RoboDK station: ConvertMoveC.rdk

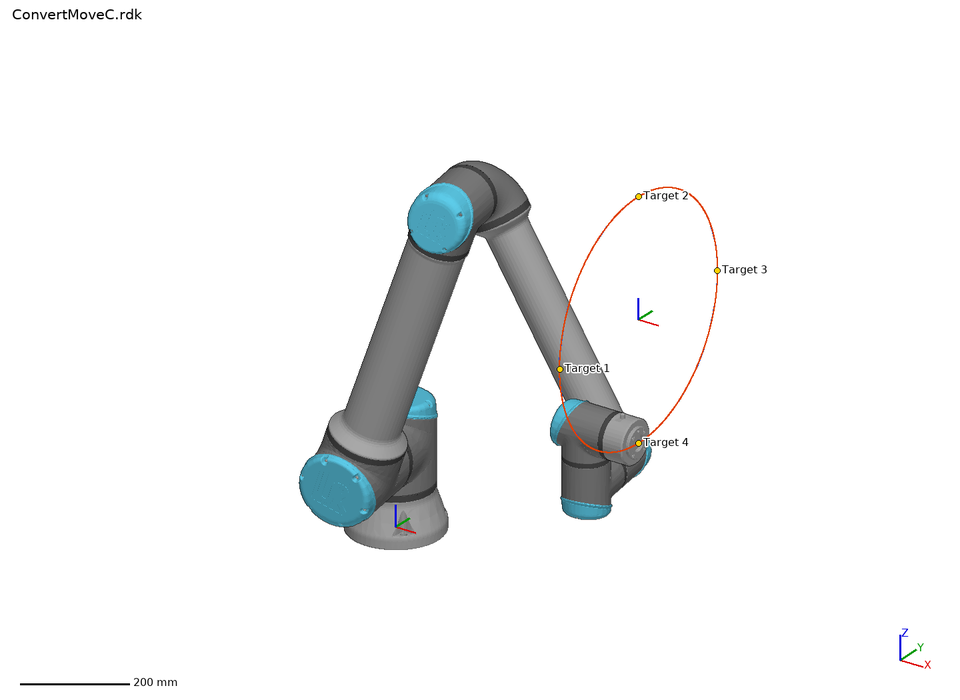
[picture v0: the station drawn from its stored meshes, robots at their saved joint values, targets as dots, program paths as lines]
Station ConvertMoveC (saved by RoboDK 5.5.2). Poses are relative to the parent item; angles as X-Y-Z fixed-axis rotations.
Station parameters (name, value as stored): ProgUtilities-Settings
  - frame UR10e Base at (0, 0, 0) mm
    - robot UR10e: 6 axes, payload 10 kg, reach 1300 mm, repeatability 0.05 mm, weight 28.9 kg
        modified DH rows (alpha deg, a mm, theta deg, d mm): 0, 0, 0, 180.7; 90, 0, 180, 0; 0, 612.6, 0, 0; 0, 571.335, 0, 174.15; -90, 0, 0, 119.85; 90, 0, 180, 116.55
        joint limits [-360, -360, -360, -360, -360, -360] to [360, 360, 360, 360, 360, 360]; home [0, -90, -90, 0, 90, 0]; saved at [8.78, -108.762, -132.424, 61.186, 81.22, 0]
    - frame Frame 2 at (610, -100, 630) mm
      - target Target 1 (Cartesian target) at (0, -250, 0) mm, rotated rx -90 ry 0 rz -90 deg; joints [-18.618, -97.519, -111.584, 29.103, 108.618, 0] of UR10e
      - target Target 2 (Cartesian target) at (0, 0, 250) mm, rotated rx -90 ry 0 rz -90 deg; joints [8.78, -80.759, -101.769, 2.528, 81.22, 0] of UR10e
      - target Target 3 (Cartesian target) at (0, 250, 0) mm, rotated rx -90 ry 0 rz -90 deg; joints [36.643, -88.986, -120.711, 29.698, 53.357, 0] of UR10e
      - target Target 4 (Cartesian target) at (0, 0, -250) mm, rotated rx -90 ry 0 rz -90 deg; joints [8.78, -108.762, -132.424, 61.186, 81.22, 0] of UR10e
  - program Prog1 (4 instructions, listed below)
  - program Prog1 Linear MoveC (1580 instructions, listed below)
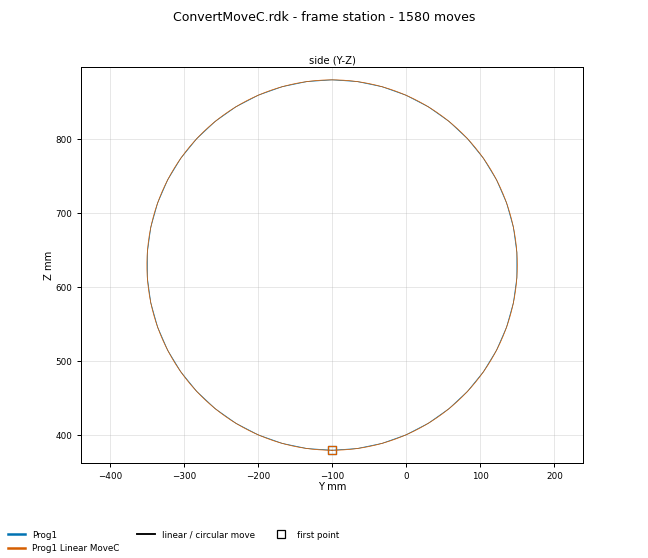
[picture p0: tool path of ConvertMoveC.rdk in frame station, 1580 of 1580 moves have a stored position in this frame; points joined in program order, loops and branches not executed]

--- program Prog1 (robot UR10e) ---
  Set Ref.: Frame 2
  MoveJ (Target 4)
  MoveC (Target 1, Target 2)
  MoveC (Target 3, Target 4)

--- program Prog1 Linear MoveC (robot UR10e) ---
  Set Ref.: Frame 2
  MoveJ (Target 4) to (0, 0, -250) mm, rotated rx -90 ry 0 rz -90 deg; joints [8.78, -108.762, -132.424, 61.186, 81.22, 0]
  MoveC (Target 1, Target 2)
  MoveL 3 to (0, 0, -250) mm, rotated rx -90 ry 0 rz -90 deg; joints [8.78, -108.762, -132.424, 61.186, 81.22, 0]
  MoveL 4 to (0, 0, -250) mm, rotated rx -90 ry 0 rz -90 deg; joints [8.78, -108.762, -132.424, 61.186, 81.22, 0]
  MoveL 5 to (0, -1, -250) mm, rotated rx -90 ry 0 rz -90 deg; joints [8.66, -108.775, -132.401, 61.176, 81.34, 0]
  MoveL 6 to (0, -2, -249.99) mm, rotated rx -90 ry 0 rz -90 deg; joints [8.541, -108.787, -132.379, 61.166, 81.459, 0]
  MoveL 7 to (0, -3, -249.98) mm, rotated rx -90 ry 0 rz -90 deg; joints [8.421, -108.8, -132.356, 61.156, 81.579, 0]
  MoveL 8 to (0, -4, -249.97) mm, rotated rx -90 ry 0 rz -90 deg; joints [8.301, -108.811, -132.333, 61.144, 81.699, 0]
  MoveL 9 to (0, -5, -249.95) mm, rotated rx -90 ry 0 rz -90 deg; joints [8.182, -108.823, -132.309, 61.132, 81.819, 0]
  MoveL 10 to (0, -5.99, -249.93) mm, rotated rx -90 ry 0 rz -90 deg; joints [8.062, -108.834, -132.286, 61.12, 81.938, 0]
  MoveL 11 to (0, -6.99, -249.9) mm, rotated rx -90 ry 0 rz -90 deg; joints [7.942, -108.845, -132.262, 61.107, 82.058, 0]
  MoveL 12 to (0, -7.99, -249.87) mm, rotated rx -90 ry 0 rz -90 deg; joints [7.823, -108.855, -132.237, 61.093, 82.177, 0]
  MoveL 13 to (0, -8.99, -249.84) mm, rotated rx -90 ry 0 rz -90 deg; joints [7.703, -108.866, -132.213, 61.078, 82.297, 0]
  MoveL 14 to (0, -9.99, -249.8) mm, rotated rx -90 ry 0 rz -90 deg; joints [7.584, -108.875, -132.188, 61.063, 82.416, 0]
  MoveL 15 to (0, -10.99, -249.76) mm, rotated rx -90 ry 0 rz -90 deg; joints [7.464, -108.885, -132.163, 61.048, 82.536, 0]
  MoveL 16 to (0, -11.99, -249.71) mm, rotated rx -90 ry 0 rz -90 deg; joints [7.345, -108.894, -132.138, 61.032, 82.655, 0]
  MoveL 17 to (0, -12.98, -249.66) mm, rotated rx -90 ry 0 rz -90 deg; joints [7.225, -108.903, -132.112, 61.015, 82.775, 0]
  MoveL 18 to (0, -13.98, -249.61) mm, rotated rx -90 ry 0 rz -90 deg; joints [7.106, -108.912, -132.086, 60.998, 82.894, 0]
  MoveL 19 to (0, -14.98, -249.55) mm, rotated rx -90 ry 0 rz -90 deg; joints [6.987, -108.92, -132.06, 60.98, 83.013, 0]
  MoveL 20 to (0, -15.98, -249.49) mm, rotated rx -90 ry 0 rz -90 deg; joints [6.868, -108.928, -132.033, 60.961, 83.132, 0]
  MoveL 21 to (0, -16.97, -249.42) mm, rotated rx -90 ry 0 rz -90 deg; joints [6.749, -108.936, -132.007, 60.942, 83.251, 0]
  MoveL 22 to (0, -17.97, -249.35) mm, rotated rx -90 ry 0 rz -90 deg; joints [6.629, -108.943, -131.98, 60.923, 83.371, 0]
  MoveL 23 to (0, -18.97, -249.28) mm, rotated rx -90 ry 0 rz -90 deg; joints [6.51, -108.95, -131.952, 60.902, 83.49, 0]
  MoveL 24 to (0, -19.96, -249.2) mm, rotated rx -90 ry 0 rz -90 deg; joints [6.392, -108.957, -131.925, 60.881, 83.608, 0]
  MoveL 25 to (0, -20.96, -249.12) mm, rotated rx -90 ry 0 rz -90 deg; joints [6.273, -108.963, -131.897, 60.86, 83.727, 0]
  MoveL 26 to (0, -21.95, -249.03) mm, rotated rx -90 ry 0 rz -90 deg; joints [6.154, -108.969, -131.869, 60.838, 83.846, 0]
  MoveL 27 to (0, -22.95, -248.94) mm, rotated rx -90 ry 0 rz -90 deg; joints [6.035, -108.975, -131.84, 60.815, 83.965, 0]
  MoveL 28 to (0, -23.94, -248.85) mm, rotated rx -90 ry 0 rz -90 deg; joints [5.917, -108.981, -131.812, 60.792, 84.083, 0]
  MoveL 29 to (0, -24.94, -248.75) mm, rotated rx -90 ry 0 rz -90 deg; joints [5.798, -108.986, -131.783, 60.769, 84.202, 0]
  MoveL 30 to (0, -25.93, -248.65) mm, rotated rx -90 ry 0 rz -90 deg; joints [5.68, -108.991, -131.754, 60.744, 84.32, 0]
  MoveL 31 to (0, -26.93, -248.55) mm, rotated rx -90 ry 0 rz -90 deg; joints [5.561, -108.995, -131.724, 60.719, 84.439, 0]
  MoveL 32 to (0, -27.92, -248.44) mm, rotated rx -90 ry 0 rz -90 deg; joints [5.443, -108.999, -131.695, 60.694, 84.557, 0]
  MoveL 33 to (0, -28.91, -248.32) mm, rotated rx -90 ry 0 rz -90 deg; joints [5.325, -109.003, -131.665, 60.668, 84.675, 0]
  MoveL 34 to (0, -29.91, -248.2) mm, rotated rx -90 ry 0 rz -90 deg; joints [5.207, -109.007, -131.634, 60.641, 84.793, 0]
  MoveL 35 to (0, -30.9, -248.08) mm, rotated rx -90 ry 0 rz -90 deg; joints [5.089, -109.01, -131.604, 60.614, 84.911, 0]
  MoveL 36 to (0, -31.89, -247.96) mm, rotated rx -90 ry 0 rz -90 deg; joints [4.971, -109.013, -131.573, 60.586, 85.029, 0]
  MoveL 37 to (0, -32.88, -247.83) mm, rotated rx -90 ry 0 rz -90 deg; joints [4.853, -109.016, -131.542, 60.558, 85.147, 0]
  MoveL 38 to (0, -33.87, -247.7) mm, rotated rx -90 ry 0 rz -90 deg; joints [4.736, -109.018, -131.511, 60.529, 85.265, 0]
  MoveL 39 to (0, -34.86, -247.56) mm, rotated rx -90 ry 0 rz -90 deg; joints [4.618, -109.02, -131.479, 60.5, 85.382, 0]
  MoveL 40 to (0, -35.85, -247.42) mm, rotated rx -90 ry 0 rz -90 deg; joints [4.501, -109.022, -131.448, 60.47, 85.499, 0]
  MoveL 41 to (0, -36.84, -247.27) mm, rotated rx -90 ry 0 rz -90 deg; joints [4.383, -109.023, -131.415, 60.439, 85.617, 0]
  MoveL 42 to (0, -37.83, -247.12) mm, rotated rx -90 ry 0 rz -90 deg; joints [4.266, -109.025, -131.383, 60.408, 85.734, 0]
  MoveL 43 to (0, -38.81, -246.97) mm, rotated rx -90 ry 0 rz -90 deg; joints [4.149, -109.025, -131.351, 60.376, 85.851, 0]
  MoveL 44 to (0, -39.8, -246.81) mm, rotated rx -90 ry 0 rz -90 deg; joints [4.032, -109.026, -131.318, 60.344, 85.968, 0]
  MoveL 45 to (0, -40.79, -246.65) mm, rotated rx -90 ry 0 rz -90 deg; joints [3.915, -109.026, -131.285, 60.311, 86.085, 0]
  MoveL 46 to (0, -41.77, -246.49) mm, rotated rx -90 ry 0 rz -90 deg; joints [3.799, -109.026, -131.251, 60.278, 86.201, 0]
  MoveL 47 to (0, -42.76, -246.32) mm, rotated rx -90 ry 0 rz -90 deg; joints [3.682, -109.026, -131.218, 60.244, 86.318, 0]
  MoveL 48 to (0, -43.74, -246.14) mm, rotated rx -90 ry 0 rz -90 deg; joints [3.566, -109.025, -131.184, 60.209, 86.434, 0]
  MoveL 49 to (0, -44.72, -245.97) mm, rotated rx -90 ry 0 rz -90 deg; joints [3.449, -109.024, -131.15, 60.174, 86.551, 0]
  MoveL 50 to (0, -45.71, -245.79) mm, rotated rx -90 ry 0 rz -90 deg; joints [3.333, -109.023, -131.116, 60.139, 86.667, 0]
  MoveL 51 to (0, -46.69, -245.6) mm, rotated rx -90 ry 0 rz -90 deg; joints [3.217, -109.021, -131.081, 60.103, 86.783, 0]
  MoveL 52 to (0, -47.67, -245.41) mm, rotated rx -90 ry 0 rz -90 deg; joints [3.101, -109.02, -131.046, 60.066, 86.899, 0]
  MoveL 53 to (0, -48.65, -245.22) mm, rotated rx -90 ry 0 rz -90 deg; joints [2.986, -109.017, -131.011, 60.029, 87.014, 0]
  MoveL 54 to (0, -49.63, -245.02) mm, rotated rx -90 ry 0 rz -90 deg; joints [2.87, -109.015, -130.976, 59.991, 87.13, 0]
  MoveL 55 to (0, -50.61, -244.82) mm, rotated rx -90 ry 0 rz -90 deg; joints [2.755, -109.012, -130.941, 59.953, 87.245, 0]
  MoveL 56 to (0, -51.59, -244.62) mm, rotated rx -90 ry 0 rz -90 deg; joints [2.639, -109.009, -130.905, 59.914, 87.361, 0]
  MoveL 57 to (0, -52.56, -244.41) mm, rotated rx -90 ry 0 rz -90 deg; joints [2.524, -109.006, -130.869, 59.875, 87.476, 0]
  MoveL 58 to (0, -53.54, -244.2) mm, rotated rx -90 ry 0 rz -90 deg; joints [2.409, -109.002, -130.833, 59.835, 87.591, 0]
  MoveL 59 to (0, -54.52, -243.98) mm, rotated rx -90 ry 0 rz -90 deg; joints [2.295, -108.999, -130.796, 59.795, 87.705, 0]
  MoveL 60 to (0, -55.49, -243.76) mm, rotated rx -90 ry 0 rz -90 deg; joints [2.18, -108.994, -130.759, 59.754, 87.82, 0]
  MoveL 61 to (0, -56.46, -243.54) mm, rotated rx -90 ry 0 rz -90 deg; joints [2.066, -108.99, -130.722, 59.712, 87.934, 0]
  MoveL 62 to (0, -57.44, -243.31) mm, rotated rx -90 ry 0 rz -90 deg; joints [1.951, -108.985, -130.685, 59.67, 88.049, 0]
  MoveL 63 to (0, -58.41, -243.08) mm, rotated rx -90 ry 0 rz -90 deg; joints [1.837, -108.98, -130.648, 59.628, 88.163, 0]
  MoveL 64 to (0, -59.38, -242.85) mm, rotated rx -90 ry 0 rz -90 deg; joints [1.723, -108.975, -130.61, 59.585, 88.277, 0]
  MoveL 65 to (0, -60.35, -242.61) mm, rotated rx -90 ry 0 rz -90 deg; joints [1.61, -108.969, -130.572, 59.541, 88.39, 0]
  MoveL 66 to (0, -61.32, -242.36) mm, rotated rx -90 ry 0 rz -90 deg; joints [1.496, -108.963, -130.534, 59.497, 88.504, 0]
  MoveL 67 to (0, -62.29, -242.12) mm, rotated rx -90 ry 0 rz -90 deg; joints [1.383, -108.957, -130.496, 59.453, 88.617, 0]
  MoveL 68 to (0, -63.26, -241.87) mm, rotated rx -90 ry 0 rz -90 deg; joints [1.27, -108.951, -130.457, 59.408, 88.73, 0]
  MoveL 69 to (0, -64.22, -241.61) mm, rotated rx -90 ry 0 rz -90 deg; joints [1.157, -108.944, -130.418, 59.362, 88.843, 0]
  MoveL 70 to (0, -65.19, -241.35) mm, rotated rx -90 ry 0 rz -90 deg; joints [1.044, -108.937, -130.379, 59.316, 88.956, 0]
  MoveL 71 to (0, -66.15, -241.09) mm, rotated rx -90 ry 0 rz -90 deg; joints [0.931, -108.93, -130.34, 59.27, 89.069, 0]
  MoveL 72 to (0, -67.11, -240.82) mm, rotated rx -90 ry 0 rz -90 deg; joints [0.819, -108.922, -130.3, 59.222, 89.181, 0]
  MoveL 73 to (0, -68.08, -240.55) mm, rotated rx -90 ry 0 rz -90 deg; joints [0.707, -108.914, -130.261, 59.175, 89.293, 0]
  MoveL 74 to (0, -69.04, -240.28) mm, rotated rx -90 ry 0 rz -90 deg; joints [0.595, -108.906, -130.221, 59.127, 89.405, 0]
  MoveL 75 to (0, -70, -240) mm, rotated rx -90 ry 0 rz -90 deg; joints [0.483, -108.898, -130.18, 59.078, 89.517, 0]
  MoveL 76 to (0, -70.96, -239.72) mm, rotated rx -90 ry 0 rz -90 deg; joints [0.371, -108.889, -130.14, 59.029, 89.629, 0]
  MoveL 77 to (0, -71.91, -239.43) mm, rotated rx -90 ry 0 rz -90 deg; joints [0.26, -108.88, -130.099, 58.98, 89.74, 0]
  MoveL 78 to (0, -72.87, -239.14) mm, rotated rx -90 ry 0 rz -90 deg; joints [0.149, -108.871, -130.059, 58.929, 89.851, 0]
  MoveL 79 to (0, -73.83, -238.85) mm, rotated rx -90 ry 0 rz -90 deg; joints [0.038, -108.861, -130.017, 58.879, 89.962, 0]
  MoveL 80 to (0, -74.78, -238.55) mm, rotated rx -90 ry 0 rz -90 deg; joints [-0.073, -108.852, -129.976, 58.828, 90.073, 0]
  MoveL 81 to (0, -75.73, -238.25) mm, rotated rx -90 ry 0 rz -90 deg; joints [-0.184, -108.842, -129.935, 58.776, 90.184, 0]
  MoveL 82 to (0, -76.68, -237.95) mm, rotated rx -90 ry 0 rz -90 deg; joints [-0.294, -108.831, -129.893, 58.724, 90.294, 0]
  MoveL 83 to (0, -77.63, -237.64) mm, rotated rx -90 ry 0 rz -90 deg; joints [-0.404, -108.821, -129.851, 58.672, 90.404, 0]
  MoveL 84 to (0, -78.58, -237.33) mm, rotated rx -90 ry 0 rz -90 deg; joints [-0.514, -108.81, -129.809, 58.619, 90.514, 0]
  MoveL 85 to (0, -79.53, -237.01) mm, rotated rx -90 ry 0 rz -90 deg; joints [-0.624, -108.799, -129.766, 58.565, 90.624, 0]
  MoveL 86 to (0, -80.48, -236.69) mm, rotated rx -90 ry 0 rz -90 deg; joints [-0.733, -108.788, -129.724, 58.511, 90.733, 0]
  MoveL 87 to (0, -81.42, -236.37) mm, rotated rx -90 ry 0 rz -90 deg; joints [-0.842, -108.776, -129.681, 58.457, 90.842, 0]
  MoveL 88 to (0, -82.37, -236.04) mm, rotated rx -90 ry 0 rz -90 deg; joints [-0.951, -108.764, -129.638, 58.402, 90.951, 0]
  MoveL 89 to (0, -83.31, -235.71) mm, rotated rx -90 ry 0 rz -90 deg; joints [-1.06, -108.752, -129.595, 58.347, 91.06, 0]
  MoveL 90 to (0, -84.25, -235.38) mm, rotated rx -90 ry 0 rz -90 deg; joints [-1.169, -108.74, -129.551, 58.291, 91.169, 0]
  MoveL 91 to (0, -85.19, -235.04) mm, rotated rx -90 ry 0 rz -90 deg; joints [-1.277, -108.727, -129.508, 58.235, 91.277, 0]
  MoveL 92 to (0, -86.13, -234.69) mm, rotated rx -90 ry 0 rz -90 deg; joints [-1.385, -108.714, -129.464, 58.178, 91.385, 0]
  MoveL 93 to (0, -87.07, -234.35) mm, rotated rx -90 ry 0 rz -90 deg; joints [-1.493, -108.701, -129.42, 58.121, 91.493, 0]
  MoveL 94 to (0, -88, -234) mm, rotated rx -90 ry 0 rz -90 deg; joints [-1.6, -108.687, -129.376, 58.063, 91.6, 0]
  MoveL 95 to (0, -88.94, -233.64) mm, rotated rx -90 ry 0 rz -90 deg; joints [-1.708, -108.674, -129.331, 58.005, 91.708, 0]
  MoveL 96 to (0, -89.87, -233.29) mm, rotated rx -90 ry 0 rz -90 deg; joints [-1.815, -108.66, -129.287, 57.946, 91.815, 0]
  MoveL 97 to (0, -90.8, -232.93) mm, rotated rx -90 ry 0 rz -90 deg; joints [-1.922, -108.646, -129.242, 57.887, 91.922, 0]
  MoveL 98 to (0, -91.73, -232.56) mm, rotated rx -90 ry 0 rz -90 deg; joints [-2.028, -108.631, -129.197, 57.828, 92.028, 0]
  MoveL 99 to (0, -92.66, -232.19) mm, rotated rx -90 ry 0 rz -90 deg; joints [-2.135, -108.617, -129.151, 57.768, 92.135, 0]
  MoveL 100 to (0, -93.59, -231.82) mm, rotated rx -90 ry 0 rz -90 deg; joints [-2.241, -108.602, -129.106, 57.708, 92.241, 0]
  MoveL 101 to (0, -94.52, -231.44) mm, rotated rx -90 ry 0 rz -90 deg; joints [-2.346, -108.587, -129.06, 57.647, 92.346, 0]
  MoveL 102 to (0, -95.44, -231.07) mm, rotated rx -90 ry 0 rz -90 deg; joints [-2.452, -108.571, -129.014, 57.586, 92.452, 0]
  MoveL 103 to (0, -96.36, -230.68) mm, rotated rx -90 ry 0 rz -90 deg; joints [-2.557, -108.555, -128.968, 57.524, 92.557, 0]
  MoveL 104 to (0, -97.28, -230.3) mm, rotated rx -90 ry 0 rz -90 deg; joints [-2.662, -108.54, -128.922, 57.462, 92.662, 0]
  MoveL 105 to (0, -98.2, -229.9) mm, rotated rx -90 ry 0 rz -90 deg; joints [-2.767, -108.523, -128.876, 57.399, 92.767, 0]
  MoveL 106 to (0, -99.12, -229.51) mm, rotated rx -90 ry 0 rz -90 deg; joints [-2.872, -108.507, -128.829, 57.336, 92.872, 0]
  MoveL 107 to (0, -100.04, -229.11) mm, rotated rx -90 ry 0 rz -90 deg; joints [-2.976, -108.49, -128.782, 57.273, 92.976, 0]
  MoveL 108 to (0, -100.95, -228.71) mm, rotated rx -90 ry 0 rz -90 deg; joints [-3.08, -108.474, -128.735, 57.209, 93.08, 0]
  MoveL 109 to (0, -101.87, -228.31) mm, rotated rx -90 ry 0 rz -90 deg; joints [-3.184, -108.456, -128.688, 57.145, 93.184, 0]
  MoveL 110 to (0, -102.78, -227.9) mm, rotated rx -90 ry 0 rz -90 deg; joints [-3.287, -108.439, -128.641, 57.08, 93.287, 0]
  MoveL 111 to (0, -103.69, -227.48) mm, rotated rx -90 ry 0 rz -90 deg; joints [-3.39, -108.422, -128.593, 57.015, 93.39, 0]
  MoveL 112 to (0, -104.6, -227.07) mm, rotated rx -90 ry 0 rz -90 deg; joints [-3.493, -108.404, -128.546, 56.949, 93.493, 0]
  MoveL 113 to (0, -105.5, -226.65) mm, rotated rx -90 ry 0 rz -90 deg; joints [-3.596, -108.386, -128.498, 56.883, 93.596, 0]
  MoveL 114 to (0, -106.41, -226.22) mm, rotated rx -90 ry 0 rz -90 deg; joints [-3.698, -108.367, -128.45, 56.817, 93.698, 0]
  MoveL 115 to (0, -107.31, -225.8) mm, rotated rx -90 ry 0 rz -90 deg; joints [-3.8, -108.349, -128.401, 56.75, 93.8, 0]
  MoveL 116 to (0, -108.21, -225.37) mm, rotated rx -90 ry 0 rz -90 deg; joints [-3.902, -108.33, -128.353, 56.683, 93.902, 0]
  MoveL 117 to (0, -109.11, -224.93) mm, rotated rx -90 ry 0 rz -90 deg; joints [-4.004, -108.311, -128.304, 56.615, 94.004, 0]
  MoveL 118 to (0, -110.01, -224.49) mm, rotated rx -90 ry 0 rz -90 deg; joints [-4.105, -108.292, -128.255, 56.547, 94.105, 0]
  MoveL 119 to (0, -110.91, -224.05) mm, rotated rx -90 ry 0 rz -90 deg; joints [-4.206, -108.273, -128.206, 56.479, 94.206, 0]
  MoveL 120 to (0, -111.8, -223.61) mm, rotated rx -90 ry 0 rz -90 deg; joints [-4.307, -108.253, -128.157, 56.41, 94.307, 0]
  MoveL 121 to (0, -112.7, -223.16) mm, rotated rx -90 ry 0 rz -90 deg; joints [-4.407, -108.233, -128.108, 56.341, 94.407, 0]
  MoveL 122 to (0, -113.59, -222.71) mm, rotated rx -90 ry 0 rz -90 deg; joints [-4.507, -108.213, -128.058, 56.271, 94.507, 0]
  MoveL 123 to (0, -114.48, -222.25) mm, rotated rx -90 ry 0 rz -90 deg; joints [-4.607, -108.193, -128.009, 56.201, 94.607, 0]
  MoveL 124 to (0, -115.36, -221.79) mm, rotated rx -90 ry 0 rz -90 deg; joints [-4.706, -108.172, -127.959, 56.131, 94.706, 0]
  MoveL 125 to (0, -116.25, -221.33) mm, rotated rx -90 ry 0 rz -90 deg; joints [-4.806, -108.151, -127.909, 56.06, 94.806, 0]
  MoveL 126 to (0, -117.13, -220.86) mm, rotated rx -90 ry 0 rz -90 deg; joints [-4.905, -108.13, -127.859, 55.989, 94.905, 0]
  MoveL 127 to (0, -118.01, -220.39) mm, rotated rx -90 ry 0 rz -90 deg; joints [-5.003, -108.109, -127.808, 55.917, 95.003, 0]
  MoveL 128 to (0, -118.89, -219.92) mm, rotated rx -90 ry 0 rz -90 deg; joints [-5.101, -108.088, -127.758, 55.846, 95.101, 0]
  MoveL 129 to (0, -119.77, -219.44) mm, rotated rx -90 ry 0 rz -90 deg; joints [-5.199, -108.066, -127.707, 55.773, 95.2, 0]
  MoveL 130 to (0, -120.65, -218.96) mm, rotated rx -90 ry 0 rz -90 deg; joints [-5.297, -108.044, -127.656, 55.701, 95.297, 0]
  MoveL 131 to (0, -121.52, -218.48) mm, rotated rx -90 ry 0 rz -90 deg; joints [-5.395, -108.022, -127.605, 55.627, 95.395, 0]
  MoveL 132 to (0, -122.39, -217.99) mm, rotated rx -90 ry 0 rz -90 deg; joints [-5.492, -108, -127.554, 55.554, 95.492, 0]
  MoveL 133 to (0, -123.27, -217.5) mm, rotated rx -90 ry 0 rz -90 deg; joints [-5.589, -107.978, -127.503, 55.48, 95.589, 0]
  MoveL 134 to (0, -124.13, -217) mm, rotated rx -90 ry 0 rz -90 deg; joints [-5.685, -107.955, -127.451, 55.406, 95.685, 0]
  MoveL 135 to (0, -125, -216.51) mm, rotated rx -90 ry 0 rz -90 deg; joints [-5.781, -107.932, -127.399, 55.331, 95.781, 0]
  MoveL 136 to (0, -125.86, -216.01) mm, rotated rx -90 ry 0 rz -90 deg; joints [-5.877, -107.909, -127.348, 55.256, 95.877, 0]
  MoveL 137 to (0, -126.73, -215.5) mm, rotated rx -90 ry 0 rz -90 deg; joints [-5.973, -107.886, -127.296, 55.181, 95.973, 0]
  MoveL 138 to (0, -127.59, -214.99) mm, rotated rx -90 ry 0 rz -90 deg; joints [-6.068, -107.862, -127.243, 55.106, 96.068, 0]
  MoveL 139 to (0, -128.45, -214.48) mm, rotated rx -90 ry 0 rz -90 deg; joints [-6.163, -107.838, -127.191, 55.03, 96.163, 0]
  MoveL 140 to (0, -129.3, -213.97) mm, rotated rx -90 ry 0 rz -90 deg; joints [-6.258, -107.815, -127.139, 54.953, 96.258, 0]
  MoveL 141 to (0, -130.16, -213.45) mm, rotated rx -90 ry 0 rz -90 deg; joints [-6.352, -107.79, -127.086, 54.876, 96.352, 0]
  MoveL 142 to (0, -131.01, -212.92) mm, rotated rx -90 ry 0 rz -90 deg; joints [-6.446, -107.766, -127.033, 54.799, 96.446, 0]
  MoveL 143 to (0, -131.86, -212.4) mm, rotated rx -90 ry 0 rz -90 deg; joints [-6.54, -107.742, -126.98, 54.722, 96.54, 0]
  MoveL 144 to (0, -132.71, -211.87) mm, rotated rx -90 ry 0 rz -90 deg; joints [-6.633, -107.717, -126.927, 54.644, 96.633, 0]
  MoveL 145 to (0, -133.55, -211.34) mm, rotated rx -90 ry 0 rz -90 deg; joints [-6.726, -107.692, -126.874, 54.566, 96.726, 0]
  MoveL 146 to (0, -134.4, -210.8) mm, rotated rx -90 ry 0 rz -90 deg; joints [-6.819, -107.667, -126.821, 54.488, 96.819, 0]
  MoveL 147 to (0, -135.24, -210.26) mm, rotated rx -90 ry 0 rz -90 deg; joints [-6.911, -107.642, -126.767, 54.409, 96.911, 0]
  MoveL 148 to (0, -136.08, -209.72) mm, rotated rx -90 ry 0 rz -90 deg; joints [-7.003, -107.616, -126.714, 54.33, 97.003, 0]
  MoveL 149 to (0, -136.91, -209.18) mm, rotated rx -90 ry 0 rz -90 deg; joints [-7.095, -107.59, -126.66, 54.25, 97.095, 0]
  MoveL 150 to (0, -137.75, -208.63) mm, rotated rx -90 ry 0 rz -90 deg; joints [-7.187, -107.565, -126.606, 54.171, 97.187, 0]
  MoveL 151 to (0, -138.58, -208.08) mm, rotated rx -90 ry 0 rz -90 deg; joints [-7.278, -107.538, -126.552, 54.09, 97.278, 0]
  MoveL 152 to (0, -139.41, -207.52) mm, rotated rx -90 ry 0 rz -90 deg; joints [-7.368, -107.512, -126.498, 54.01, 97.368, 0]
  MoveL 153 to (0, -140.24, -206.96) mm, rotated rx -90 ry 0 rz -90 deg; joints [-7.459, -107.486, -126.443, 53.929, 97.459, 0]
  MoveL 154 to (0, -141.07, -206.4) mm, rotated rx -90 ry 0 rz -90 deg; joints [-7.549, -107.459, -126.389, 53.848, 97.549, 0]
  MoveL 155 to (0, -141.89, -205.83) mm, rotated rx -90 ry 0 rz -90 deg; joints [-7.639, -107.432, -126.334, 53.767, 97.639, 0]
  MoveL 156 to (0, -142.71, -205.26) mm, rotated rx -90 ry 0 rz -90 deg; joints [-7.728, -107.405, -126.279, 53.685, 97.728, 0]
  MoveL 157 to (0, -143.53, -204.69) mm, rotated rx -90 ry 0 rz -90 deg; joints [-7.817, -107.378, -126.225, 53.603, 97.817, 0]
  MoveL 158 to (0, -144.35, -204.12) mm, rotated rx -90 ry 0 rz -90 deg; joints [-7.906, -107.351, -126.17, 53.52, 97.906, 0]
  MoveL 159 to (0, -145.16, -203.54) mm, rotated rx -90 ry 0 rz -90 deg; joints [-7.995, -107.323, -126.114, 53.438, 97.995, 0]
  MoveL 160 to (0, -145.97, -202.96) mm, rotated rx -90 ry 0 rz -90 deg; joints [-8.083, -107.295, -126.059, 53.355, 98.083, 0]
  MoveL 161 to (0, -146.78, -202.37) mm, rotated rx -90 ry 0 rz -90 deg; joints [-8.171, -107.268, -126.004, 53.271, 98.171, 0]
  MoveL 162 to (0, -147.59, -201.78) mm, rotated rx -90 ry 0 rz -90 deg; joints [-8.258, -107.239, -125.948, 53.188, 98.258, 0]
  MoveL 163 to (0, -148.4, -201.19) mm, rotated rx -90 ry 0 rz -90 deg; joints [-8.345, -107.211, -125.892, 53.104, 98.345, 0]
  MoveL 164 to (0, -149.2, -200.6) mm, rotated rx -90 ry 0 rz -90 deg; joints [-8.432, -107.183, -125.837, 53.019, 98.432, 0]
  MoveL 165 to (0, -150, -200) mm, rotated rx -90 ry 0 rz -90 deg; joints [-8.518, -107.154, -125.781, 52.935, 98.518, 0]
  MoveL 166 to (0, -150.8, -199.4) mm, rotated rx -90 ry 0 rz -90 deg; joints [-8.605, -107.125, -125.725, 52.85, 98.605, 0]
  MoveL 167 to (0, -151.6, -198.79) mm, rotated rx -90 ry 0 rz -90 deg; joints [-8.69, -107.096, -125.669, 52.765, 98.69, 0]
  MoveL 168 to (0, -152.39, -198.19) mm, rotated rx -90 ry 0 rz -90 deg; joints [-8.776, -107.067, -125.612, 52.68, 98.776, 0]
  MoveL 169 to (0, -153.18, -197.58) mm, rotated rx -90 ry 0 rz -90 deg; joints [-8.861, -107.038, -125.556, 52.594, 98.861, 0]
  MoveL 170 to (0, -153.97, -196.96) mm, rotated rx -90 ry 0 rz -90 deg; joints [-8.945, -107.008, -125.499, 52.508, 98.946, 0]
  MoveL 171 to (0, -154.75, -196.34) mm, rotated rx -90 ry 0 rz -90 deg; joints [-9.03, -106.979, -125.443, 52.421, 99.03, 0]
  MoveL 172 to (0, -155.54, -195.72) mm, rotated rx -90 ry 0 rz -90 deg; joints [-9.114, -106.949, -125.386, 52.335, 99.114, 0]
  MoveL 173 to (0, -156.32, -195.1) mm, rotated rx -90 ry 0 rz -90 deg; joints [-9.198, -106.919, -125.329, 52.248, 99.198, 0]
  MoveL 174 to (0, -157.1, -194.48) mm, rotated rx -90 ry 0 rz -90 deg; joints [-9.281, -106.889, -125.272, 52.161, 99.281, 0]
  MoveL 175 to (0, -157.87, -193.85) mm, rotated rx -90 ry 0 rz -90 deg; joints [-9.364, -106.859, -125.215, 52.073, 99.364, 0]
  MoveL 176 to (0, -158.65, -193.21) mm, rotated rx -90 ry 0 rz -90 deg; joints [-9.447, -106.828, -125.158, 51.986, 99.447, 0]
  MoveL 177 to (0, -159.42, -192.58) mm, rotated rx -90 ry 0 rz -90 deg; joints [-9.529, -106.797, -125.1, 51.898, 99.529, 0]
  MoveL 178 to (0, -160.19, -191.94) mm, rotated rx -90 ry 0 rz -90 deg; joints [-9.611, -106.767, -125.043, 51.809, 99.611, 0]
  MoveL 179 to (0, -160.95, -191.3) mm, rotated rx -90 ry 0 rz -90 deg; joints [-9.692, -106.736, -124.985, 51.721, 99.692, 0]
  MoveL 180 to (0, -161.72, -190.65) mm, rotated rx -90 ry 0 rz -90 deg; joints [-9.774, -106.705, -124.928, 51.632, 99.774, 0]
  MoveL 181 to (0, -162.48, -190) mm, rotated rx -90 ry 0 rz -90 deg; joints [-9.855, -106.673, -124.87, 51.543, 99.855, 0]
  MoveL 182 to (0, -163.23, -189.35) mm, rotated rx -90 ry 0 rz -90 deg; joints [-9.935, -106.642, -124.812, 51.454, 99.935, 0]
  MoveL 183 to (0, -163.99, -188.7) mm, rotated rx -90 ry 0 rz -90 deg; joints [-10.015, -106.61, -124.754, 51.364, 100.015, 0]
  MoveL 184 to (0, -164.74, -188.04) mm, rotated rx -90 ry 0 rz -90 deg; joints [-10.095, -106.578, -124.696, 51.274, 100.095, 0]
  MoveL 185 to (0, -165.49, -187.38) mm, rotated rx -90 ry 0 rz -90 deg; joints [-10.175, -106.547, -124.638, 51.184, 100.175, 0]
  MoveL 186 to (0, -166.24, -186.72) mm, rotated rx -90 ry 0 rz -90 deg; joints [-10.254, -106.514, -124.579, 51.094, 100.254, 0]
  MoveL 187 to (0, -166.99, -186.05) mm, rotated rx -90 ry 0 rz -90 deg; joints [-10.333, -106.482, -124.521, 51.003, 100.333, 0]
  MoveL 188 to (0, -167.73, -185.38) mm, rotated rx -90 ry 0 rz -90 deg; joints [-10.411, -106.45, -124.462, 50.912, 100.411, 0]
  MoveL 189 to (0, -168.47, -184.71) mm, rotated rx -90 ry 0 rz -90 deg; joints [-10.489, -106.417, -124.404, 50.821, 100.489, 0]
  MoveL 190 to (0, -169.2, -184.04) mm, rotated rx -90 ry 0 rz -90 deg; joints [-10.567, -106.385, -124.345, 50.73, 100.567, 0]
  MoveL 191 to (0, -169.94, -183.36) mm, rotated rx -90 ry 0 rz -90 deg; joints [-10.644, -106.352, -124.286, 50.638, 100.644, 0]
  MoveL 192 to (0, -170.67, -182.68) mm, rotated rx -90 ry 0 rz -90 deg; joints [-10.721, -106.319, -124.227, 50.546, 100.721, 0]
  MoveL 193 to (0, -171.4, -182) mm, rotated rx -90 ry 0 rz -90 deg; joints [-10.798, -106.286, -124.168, 50.454, 100.798, 0]
  MoveL 194 to (0, -172.12, -181.31) mm, rotated rx -90 ry 0 rz -90 deg; joints [-10.874, -106.253, -124.109, 50.362, 100.874, 0]
  MoveL 195 to (0, -172.85, -180.62) mm, rotated rx -90 ry 0 rz -90 deg; joints [-10.95, -106.219, -124.05, 50.269, 100.95, 0]
  MoveL 196 to (0, -173.57, -179.93) mm, rotated rx -90 ry 0 rz -90 deg; joints [-11.025, -106.186, -123.991, 50.176, 101.025, 0]
  MoveL 197 to (0, -174.29, -179.23) mm, rotated rx -90 ry 0 rz -90 deg; joints [-11.101, -106.152, -123.931, 50.083, 101.101, 0]
  MoveL 198 to (0, -175, -178.53) mm, rotated rx -90 ry 0 rz -90 deg; joints [-11.175, -106.118, -123.872, 49.99, 101.175, 0]
  MoveL 199 to (0, -175.71, -177.83) mm, rotated rx -90 ry 0 rz -90 deg; joints [-11.25, -106.084, -123.812, 49.897, 101.25, 0]
  MoveL 200 to (0, -176.42, -177.13) mm, rotated rx -90 ry 0 rz -90 deg; joints [-11.324, -106.05, -123.753, 49.803, 101.324, 0]
  MoveL 201 to (0, -177.13, -176.42) mm, rotated rx -90 ry 0 rz -90 deg; joints [-11.398, -106.016, -123.693, 49.709, 101.398, 0]
  MoveL 202 to (0, -177.83, -175.71) mm, rotated rx -90 ry 0 rz -90 deg; joints [-11.471, -105.981, -123.633, 49.615, 101.471, 0]
  MoveL 203 to (0, -178.53, -175) mm, rotated rx -90 ry 0 rz -90 deg; joints [-11.544, -105.947, -123.573, 49.52, 101.544, 0]
  MoveL 204 to (0, -179.23, -174.29) mm, rotated rx -90 ry 0 rz -90 deg; joints [-11.617, -105.912, -123.513, 49.426, 101.617, 0]
  MoveL 205 to (0, -179.93, -173.57) mm, rotated rx -90 ry 0 rz -90 deg; joints [-11.689, -105.877, -123.453, 49.331, 101.689, 0]
  MoveL 206 to (0, -180.62, -172.85) mm, rotated rx -90 ry 0 rz -90 deg; joints [-11.761, -105.842, -123.393, 49.236, 101.761, 0]
  MoveL 207 to (0, -181.31, -172.12) mm, rotated rx -90 ry 0 rz -90 deg; joints [-11.832, -105.807, -123.333, 49.14, 101.832, 0]
  MoveL 208 to (0, -182, -171.4) mm, rotated rx -90 ry 0 rz -90 deg; joints [-11.904, -105.772, -123.273, 49.045, 101.904, 0]
  MoveL 209 to (0, -182.68, -170.67) mm, rotated rx -90 ry 0 rz -90 deg; joints [-11.974, -105.737, -123.212, 48.949, 101.974, 0]
  MoveL 210 to (0, -183.36, -169.94) mm, rotated rx -90 ry 0 rz -90 deg; joints [-12.045, -105.701, -123.152, 48.853, 102.045, 0]
  MoveL 211 to (0, -184.04, -169.2) mm, rotated rx -90 ry 0 rz -90 deg; joints [-12.115, -105.666, -123.091, 48.757, 102.115, 0]
  MoveL 212 to (0, -184.71, -168.47) mm, rotated rx -90 ry 0 rz -90 deg; joints [-12.185, -105.63, -123.031, 48.661, 102.185, 0]
  MoveL 213 to (0, -185.38, -167.73) mm, rotated rx -90 ry 0 rz -90 deg; joints [-12.254, -105.594, -122.97, 48.564, 102.254, 0]
  MoveL 214 to (0, -186.05, -166.99) mm, rotated rx -90 ry 0 rz -90 deg; joints [-12.323, -105.558, -122.909, 48.467, 102.323, 0]
  MoveL 215 to (0, -186.72, -166.24) mm, rotated rx -90 ry 0 rz -90 deg; joints [-12.392, -105.522, -122.848, 48.37, 102.392, 0]
  MoveL 216 to (0, -187.38, -165.49) mm, rotated rx -90 ry 0 rz -90 deg; joints [-12.46, -105.486, -122.787, 48.273, 102.46, 0]
  MoveL 217 to (0, -188.04, -164.74) mm, rotated rx -90 ry 0 rz -90 deg; joints [-12.528, -105.449, -122.727, 48.176, 102.528, 0]
  MoveL 218 to (0, -188.7, -163.99) mm, rotated rx -90 ry 0 rz -90 deg; joints [-12.595, -105.413, -122.666, 48.078, 102.595, 0]
  MoveL 219 to (0, -189.35, -163.23) mm, rotated rx -90 ry 0 rz -90 deg; joints [-12.662, -105.376, -122.604, 47.981, 102.662, 0]
  MoveL 220 to (0, -190, -162.48) mm, rotated rx -90 ry 0 rz -90 deg; joints [-12.729, -105.34, -122.543, 47.883, 102.729, 0]
  MoveL 221 to (0, -190.65, -161.72) mm, rotated rx -90 ry 0 rz -90 deg; joints [-12.795, -105.303, -122.482, 47.785, 102.795, 0]
  MoveL 222 to (0, -191.3, -160.95) mm, rotated rx -90 ry 0 rz -90 deg; joints [-12.861, -105.266, -122.421, 47.687, 102.861, 0]
  MoveL 223 to (0, -191.94, -160.19) mm, rotated rx -90 ry 0 rz -90 deg; joints [-12.927, -105.229, -122.359, 47.588, 102.927, 0]
  MoveL 224 to (0, -192.58, -159.42) mm, rotated rx -90 ry 0 rz -90 deg; joints [-12.992, -105.191, -122.298, 47.489, 102.992, 0]
  MoveL 225 to (0, -193.21, -158.65) mm, rotated rx -90 ry 0 rz -90 deg; joints [-13.057, -105.154, -122.236, 47.391, 103.057, 0]
  MoveL 226 to (0, -193.85, -157.87) mm, rotated rx -90 ry 0 rz -90 deg; joints [-13.122, -105.117, -122.175, 47.292, 103.122, 0]
  MoveL 227 to (0, -194.48, -157.1) mm, rotated rx -90 ry 0 rz -90 deg; joints [-13.186, -105.079, -122.113, 47.192, 103.186, 0]
  MoveL 228 to (0, -195.1, -156.32) mm, rotated rx -90 ry 0 rz -90 deg; joints [-13.25, -105.041, -122.052, 47.093, 103.25, 0]
  MoveL 229 to (0, -195.72, -155.54) mm, rotated rx -90 ry 0 rz -90 deg; joints [-13.313, -105.004, -121.99, 46.994, 103.313, 0]
  MoveL 230 to (0, -196.34, -154.75) mm, rotated rx -90 ry 0 rz -90 deg; joints [-13.376, -104.966, -121.928, 46.894, 103.376, 0]
  MoveL 231 to (0, -196.96, -153.97) mm, rotated rx -90 ry 0 rz -90 deg; joints [-13.439, -104.928, -121.866, 46.794, 103.439, 0]
  MoveL 232 to (0, -197.58, -153.18) mm, rotated rx -90 ry 0 rz -90 deg; joints [-13.501, -104.889, -121.804, 46.694, 103.501, 0]
  MoveL 233 to (0, -198.19, -152.39) mm, rotated rx -90 ry 0 rz -90 deg; joints [-13.563, -104.851, -121.743, 46.594, 103.563, 0]
  MoveL 234 to (0, -198.79, -151.6) mm, rotated rx -90 ry 0 rz -90 deg; joints [-13.624, -104.813, -121.681, 46.493, 103.625, 0]
  MoveL 235 to (0, -199.4, -150.8) mm, rotated rx -90 ry 0 rz -90 deg; joints [-13.686, -104.774, -121.619, 46.393, 103.686, 0]
  MoveL 236 to (0, -200, -150) mm, rotated rx -90 ry 0 rz -90 deg; joints [-13.746, -104.736, -121.556, 46.292, 103.746, 0]
  MoveL 237 to (0, -200.6, -149.2) mm, rotated rx -90 ry 0 rz -90 deg; joints [-13.807, -104.697, -121.494, 46.191, 103.807, 0]
  MoveL 238 to (0, -201.19, -148.4) mm, rotated rx -90 ry 0 rz -90 deg; joints [-13.867, -104.658, -121.432, 46.09, 103.867, 0]
  MoveL 239 to (0, -201.78, -147.59) mm, rotated rx -90 ry 0 rz -90 deg; joints [-13.927, -104.619, -121.37, 45.989, 103.927, 0]
  MoveL 240 to (0, -202.37, -146.78) mm, rotated rx -90 ry 0 rz -90 deg; joints [-13.986, -104.58, -121.308, 45.888, 103.986, 0]
  MoveL 241 to (0, -202.96, -145.97) mm, rotated rx -90 ry 0 rz -90 deg; joints [-14.045, -104.541, -121.245, 45.786, 104.045, 0]
  MoveL 242 to (0, -203.54, -145.16) mm, rotated rx -90 ry 0 rz -90 deg; joints [-14.103, -104.502, -121.183, 45.685, 104.103, 0]
  MoveL 243 to (0, -204.12, -144.35) mm, rotated rx -90 ry 0 rz -90 deg; joints [-14.161, -104.463, -121.12, 45.583, 104.161, 0]
  MoveL 244 to (0, -204.69, -143.53) mm, rotated rx -90 ry 0 rz -90 deg; joints [-14.219, -104.423, -121.058, 45.481, 104.219, 0]
  MoveL 245 to (0, -205.26, -142.71) mm, rotated rx -90 ry 0 rz -90 deg; joints [-14.277, -104.384, -120.996, 45.379, 104.277, 0]
  MoveL 246 to (0, -205.83, -141.89) mm, rotated rx -90 ry 0 rz -90 deg; joints [-14.334, -104.344, -120.933, 45.277, 104.334, 0]
  MoveL 247 to (0, -206.4, -141.07) mm, rotated rx -90 ry 0 rz -90 deg; joints [-14.39, -104.304, -120.87, 45.175, 104.39, 0]
  MoveL 248 to (0, -206.96, -140.24) mm, rotated rx -90 ry 0 rz -90 deg; joints [-14.447, -104.264, -120.808, 45.072, 104.447, 0]
  MoveL 249 to (0, -207.52, -139.41) mm, rotated rx -90 ry 0 rz -90 deg; joints [-14.503, -104.224, -120.745, 44.97, 104.503, 0]
  MoveL 250 to (0, -208.08, -138.58) mm, rotated rx -90 ry 0 rz -90 deg; joints [-14.558, -104.184, -120.683, 44.867, 104.558, 0]
  MoveL 251 to (0, -208.63, -137.75) mm, rotated rx -90 ry 0 rz -90 deg; joints [-14.613, -104.144, -120.62, 44.764, 104.613, 0]
  MoveL 252 to (0, -209.18, -136.91) mm, rotated rx -90 ry 0 rz -90 deg; joints [-14.668, -104.104, -120.557, 44.661, 104.668, 0]
  MoveL 253 to (0, -209.72, -136.08) mm, rotated rx -90 ry 0 rz -90 deg; joints [-14.722, -104.063, -120.494, 44.558, 104.722, 0]
  MoveL 254 to (0, -210.26, -135.24) mm, rotated rx -90 ry 0 rz -90 deg; joints [-14.776, -104.023, -120.431, 44.455, 104.776, 0]
  MoveL 255 to (0, -210.8, -134.4) mm, rotated rx -90 ry 0 rz -90 deg; joints [-14.83, -103.982, -120.369, 44.351, 104.83, 0]
  MoveL 256 to (0, -211.34, -133.55) mm, rotated rx -90 ry 0 rz -90 deg; joints [-14.883, -103.942, -120.306, 44.248, 104.883, 0]
  MoveL 257 to (0, -211.87, -132.71) mm, rotated rx -90 ry 0 rz -90 deg; joints [-14.936, -103.901, -120.243, 44.144, 104.936, 0]
  MoveL 258 to (0, -212.4, -131.86) mm, rotated rx -90 ry 0 rz -90 deg; joints [-14.989, -103.86, -120.18, 44.04, 104.989, 0]
  MoveL 259 to (0, -212.92, -131.01) mm, rotated rx -90 ry 0 rz -90 deg; joints [-15.041, -103.819, -120.117, 43.936, 105.041, 0]
  MoveL 260 to (0, -213.45, -130.16) mm, rotated rx -90 ry 0 rz -90 deg; joints [-15.093, -103.778, -120.054, 43.832, 105.093, 0]
  MoveL 261 to (0, -213.97, -129.3) mm, rotated rx -90 ry 0 rz -90 deg; joints [-15.144, -103.737, -119.991, 43.728, 105.144, 0]
  MoveL 262 to (0, -214.48, -128.45) mm, rotated rx -90 ry 0 rz -90 deg; joints [-15.195, -103.696, -119.928, 43.624, 105.195, 0]
  MoveL 263 to (0, -214.99, -127.59) mm, rotated rx -90 ry 0 rz -90 deg; joints [-15.246, -103.655, -119.865, 43.52, 105.246, 0]
  MoveL 264 to (0, -215.5, -126.73) mm, rotated rx -90 ry 0 rz -90 deg; joints [-15.296, -103.613, -119.802, 43.415, 105.296, 0]
  MoveL 265 to (0, -216.01, -125.86) mm, rotated rx -90 ry 0 rz -90 deg; joints [-15.346, -103.572, -119.739, 43.311, 105.346, 0]
  MoveL 266 to (0, -216.51, -125) mm, rotated rx -90 ry 0 rz -90 deg; joints [-15.395, -103.53, -119.676, 43.206, 105.395, 0]
  MoveL 267 to (0, -217, -124.13) mm, rotated rx -90 ry 0 rz -90 deg; joints [-15.444, -103.489, -119.612, 43.101, 105.444, 0]
  MoveL 268 to (0, -217.5, -123.27) mm, rotated rx -90 ry 0 rz -90 deg; joints [-15.493, -103.447, -119.549, 42.996, 105.493, 0]
  MoveL 269 to (0, -217.99, -122.39) mm, rotated rx -90 ry 0 rz -90 deg; joints [-15.541, -103.405, -119.486, 42.891, 105.542, 0]
  MoveL 270 to (0, -218.48, -121.52) mm, rotated rx -90 ry 0 rz -90 deg; joints [-15.589, -103.363, -119.423, 42.786, 105.589, 0]
  MoveL 271 to (0, -218.96, -120.65) mm, rotated rx -90 ry 0 rz -90 deg; joints [-15.637, -103.321, -119.36, 42.681, 105.637, 0]
  MoveL 272 to (0, -219.44, -119.77) mm, rotated rx -90 ry 0 rz -90 deg; joints [-15.684, -103.279, -119.296, 42.576, 105.684, 0]
  MoveL 273 to (0, -219.92, -118.89) mm, rotated rx -90 ry 0 rz -90 deg; joints [-15.731, -103.237, -119.233, 42.47, 105.731, 0]
  MoveL 274 to (0, -220.39, -118.01) mm, rotated rx -90 ry 0 rz -90 deg; joints [-15.778, -103.195, -119.17, 42.365, 105.778, 0]
  MoveL 275 to (0, -220.86, -117.13) mm, rotated rx -90 ry 0 rz -90 deg; joints [-15.824, -103.152, -119.107, 42.259, 105.824, 0]
  MoveL 276 to (0, -221.33, -116.25) mm, rotated rx -90 ry 0 rz -90 deg; joints [-15.869, -103.11, -119.043, 42.153, 105.869, 0]
  MoveL 277 to (0, -221.79, -115.36) mm, rotated rx -90 ry 0 rz -90 deg; joints [-15.915, -103.067, -118.98, 42.048, 105.915, 0]
  MoveL 278 to (0, -222.25, -114.48) mm, rotated rx -90 ry 0 rz -90 deg; joints [-15.96, -103.025, -118.917, 41.942, 105.96, 0]
  MoveL 279 to (0, -222.71, -113.59) mm, rotated rx -90 ry 0 rz -90 deg; joints [-16.004, -102.982, -118.854, 41.836, 106.004, 0]
  MoveL 280 to (0, -223.16, -112.7) mm, rotated rx -90 ry 0 rz -90 deg; joints [-16.048, -102.939, -118.79, 41.73, 106.049, 0]
  MoveL 281 to (0, -223.61, -111.8) mm, rotated rx -90 ry 0 rz -90 deg; joints [-16.092, -102.897, -118.727, 41.624, 106.092, 0]
  MoveL 282 to (0, -224.05, -110.91) mm, rotated rx -90 ry 0 rz -90 deg; joints [-16.136, -102.854, -118.664, 41.517, 106.136, 0]
  MoveL 283 to (0, -224.49, -110.01) mm, rotated rx -90 ry 0 rz -90 deg; joints [-16.179, -102.811, -118.6, 41.411, 106.179, 0]
  MoveL 284 to (0, -224.93, -109.11) mm, rotated rx -90 ry 0 rz -90 deg; joints [-16.221, -102.768, -118.537, 41.305, 106.222, 0]
  MoveL 285 to (0, -225.37, -108.21) mm, rotated rx -90 ry 0 rz -90 deg; joints [-16.264, -102.724, -118.474, 41.198, 106.264, 0]
  MoveL 286 to (0, -225.8, -107.31) mm, rotated rx -90 ry 0 rz -90 deg; joints [-16.306, -102.681, -118.41, 41.092, 106.306, 0]
  MoveL 287 to (0, -226.22, -106.41) mm, rotated rx -90 ry 0 rz -90 deg; joints [-16.347, -102.638, -118.347, 40.985, 106.347, 0]
  MoveL 288 to (0, -226.65, -105.5) mm, rotated rx -90 ry 0 rz -90 deg; joints [-16.388, -102.595, -118.284, 40.878, 106.388, 0]
  MoveL 289 to (0, -227.07, -104.6) mm, rotated rx -90 ry 0 rz -90 deg; joints [-16.429, -102.551, -118.22, 40.772, 106.429, 0]
  MoveL 290 to (0, -227.48, -103.69) mm, rotated rx -90 ry 0 rz -90 deg; joints [-16.47, -102.508, -118.157, 40.665, 106.47, 0]
  MoveL 291 to (0, -227.9, -102.78) mm, rotated rx -90 ry 0 rz -90 deg; joints [-16.51, -102.464, -118.094, 40.558, 106.51, 0]
  MoveL 292 to (0, -228.31, -101.87) mm, rotated rx -90 ry 0 rz -90 deg; joints [-16.549, -102.42, -118.031, 40.451, 106.549, 0]
  MoveL 293 to (0, -228.71, -100.95) mm, rotated rx -90 ry 0 rz -90 deg; joints [-16.589, -102.377, -117.967, 40.344, 106.589, 0]
  MoveL 294 to (0, -229.11, -100.04) mm, rotated rx -90 ry 0 rz -90 deg; joints [-16.628, -102.333, -117.904, 40.237, 106.628, 0]
  MoveL 295 to (0, -229.51, -99.12) mm, rotated rx -90 ry 0 rz -90 deg; joints [-16.666, -102.289, -117.841, 40.13, 106.666, 0]
  MoveL 296 to (0, -229.9, -98.2) mm, rotated rx -90 ry 0 rz -90 deg; joints [-16.704, -102.245, -117.777, 40.022, 106.704, 0]
  MoveL 297 to (0, -230.3, -97.28) mm, rotated rx -90 ry 0 rz -90 deg; joints [-16.742, -102.201, -117.714, 39.915, 106.742, 0]
  MoveL 298 to (0, -230.68, -96.36) mm, rotated rx -90 ry 0 rz -90 deg; joints [-16.779, -102.157, -117.651, 39.808, 106.779, 0]
  MoveL 299 to (0, -231.07, -95.44) mm, rotated rx -90 ry 0 rz -90 deg; joints [-16.816, -102.113, -117.588, 39.7, 106.816, 0]
  MoveL 300 to (0, -231.44, -94.52) mm, rotated rx -90 ry 0 rz -90 deg; joints [-16.853, -102.068, -117.524, 39.593, 106.853, 0]
  MoveL 301 to (0, -231.82, -93.59) mm, rotated rx -90 ry 0 rz -90 deg; joints [-16.889, -102.024, -117.461, 39.485, 106.889, 0]
  MoveL 302 to (0, -232.19, -92.66) mm, rotated rx -90 ry 0 rz -90 deg; joints [-16.925, -101.98, -117.398, 39.378, 106.925, 0]
  MoveL 303 to (0, -232.56, -91.73) mm, rotated rx -90 ry 0 rz -90 deg; joints [-16.961, -101.935, -117.335, 39.27, 106.961, 0]
  MoveL 304 to (0, -232.93, -90.8) mm, rotated rx -90 ry 0 rz -90 deg; joints [-16.996, -101.891, -117.272, 39.162, 106.996, 0]
  MoveL 305 to (0, -233.29, -89.87) mm, rotated rx -90 ry 0 rz -90 deg; joints [-17.031, -101.846, -117.208, 39.055, 107.031, 0]
  MoveL 306 to (0, -233.64, -88.94) mm, rotated rx -90 ry 0 rz -90 deg; joints [-17.065, -101.801, -117.145, 38.947, 107.065, 0]
  MoveL 307 to (0, -234, -88) mm, rotated rx -90 ry 0 rz -90 deg; joints [-17.099, -101.757, -117.082, 38.839, 107.099, 0]
  MoveL 308 to (0, -234.35, -87.07) mm, rotated rx -90 ry 0 rz -90 deg; joints [-17.133, -101.712, -117.019, 38.731, 107.133, 0]
  MoveL 309 to (0, -234.69, -86.13) mm, rotated rx -90 ry 0 rz -90 deg; joints [-17.166, -101.667, -116.956, 38.623, 107.166, 0]
  MoveL 310 to (0, -235.04, -85.19) mm, rotated rx -90 ry 0 rz -90 deg; joints [-17.199, -101.622, -116.893, 38.515, 107.199, 0]
  MoveL 311 to (0, -235.38, -84.25) mm, rotated rx -90 ry 0 rz -90 deg; joints [-17.231, -101.577, -116.83, 38.407, 107.231, 0]
  MoveL 312 to (0, -235.71, -83.31) mm, rotated rx -90 ry 0 rz -90 deg; joints [-17.263, -101.532, -116.767, 38.299, 107.263, 0]
  MoveL 313 to (0, -236.04, -82.37) mm, rotated rx -90 ry 0 rz -90 deg; joints [-17.295, -101.487, -116.704, 38.191, 107.295, 0]
  MoveL 314 to (0, -236.37, -81.42) mm, rotated rx -90 ry 0 rz -90 deg; joints [-17.326, -101.442, -116.641, 38.083, 107.326, 0]
  MoveL 315 to (0, -236.69, -80.48) mm, rotated rx -90 ry 0 rz -90 deg; joints [-17.357, -101.397, -116.578, 37.975, 107.357, 0]
  MoveL 316 to (0, -237.01, -79.53) mm, rotated rx -90 ry 0 rz -90 deg; joints [-17.388, -101.351, -116.515, 37.866, 107.388, 0]
  MoveL 317 to (0, -237.33, -78.58) mm, rotated rx -90 ry 0 rz -90 deg; joints [-17.418, -101.306, -116.452, 37.758, 107.418, 0]
  MoveL 318 to (0, -237.64, -77.63) mm, rotated rx -90 ry 0 rz -90 deg; joints [-17.448, -101.261, -116.389, 37.65, 107.448, 0]
  MoveL 319 to (0, -237.95, -76.68) mm, rotated rx -90 ry 0 rz -90 deg; joints [-17.477, -101.215, -116.326, 37.542, 107.477, 0]
  MoveL 320 to (0, -238.25, -75.73) mm, rotated rx -90 ry 0 rz -90 deg; joints [-17.506, -101.17, -116.263, 37.433, 107.507, 0]
  MoveL 321 to (0, -238.55, -74.78) mm, rotated rx -90 ry 0 rz -90 deg; joints [-17.535, -101.124, -116.201, 37.325, 107.535, 0]
  MoveL 322 to (0, -238.85, -73.83) mm, rotated rx -90 ry 0 rz -90 deg; joints [-17.564, -101.079, -116.138, 37.216, 107.564, 0]
  MoveL 323 to (0, -239.14, -72.87) mm, rotated rx -90 ry 0 rz -90 deg; joints [-17.591, -101.033, -116.075, 37.108, 107.592, 0]
  MoveL 324 to (0, -239.43, -71.91) mm, rotated rx -90 ry 0 rz -90 deg; joints [-17.619, -100.987, -116.013, 37, 107.619, 0]
  MoveL 325 to (0, -239.72, -70.96) mm, rotated rx -90 ry 0 rz -90 deg; joints [-17.646, -100.941, -115.95, 36.891, 107.646, 0]
  MoveL 326 to (0, -240, -70) mm, rotated rx -90 ry 0 rz -90 deg; joints [-17.673, -100.895, -115.887, 36.783, 107.673, 0]
  MoveL 327 to (0, -240.28, -69.04) mm, rotated rx -90 ry 0 rz -90 deg; joints [-17.7, -100.849, -115.825, 36.674, 107.7, 0]
  MoveL 328 to (0, -240.55, -68.08) mm, rotated rx -90 ry 0 rz -90 deg; joints [-17.726, -100.803, -115.762, 36.566, 107.726, 0]
  MoveL 329 to (0, -240.82, -67.11) mm, rotated rx -90 ry 0 rz -90 deg; joints [-17.751, -100.757, -115.7, 36.457, 107.751, 0]
  MoveL 330 to (0, -241.09, -66.15) mm, rotated rx -90 ry 0 rz -90 deg; joints [-17.777, -100.711, -115.637, 36.349, 107.777, 0]
  MoveL 331 to (0, -241.35, -65.19) mm, rotated rx -90 ry 0 rz -90 deg; joints [-17.802, -100.665, -115.575, 36.24, 107.802, 0]
  MoveL 332 to (0, -241.61, -64.22) mm, rotated rx -90 ry 0 rz -90 deg; joints [-17.826, -100.619, -115.512, 36.131, 107.826, 0]
  MoveL 333 to (0, -241.87, -63.26) mm, rotated rx -90 ry 0 rz -90 deg; joints [-17.85, -100.573, -115.45, 36.023, 107.85, 0]
  MoveL 334 to (0, -242.12, -62.29) mm, rotated rx -90 ry 0 rz -90 deg; joints [-17.874, -100.526, -115.388, 35.914, 107.874, 0]
  MoveL 335 to (0, -242.36, -61.32) mm, rotated rx -90 ry 0 rz -90 deg; joints [-17.898, -100.48, -115.325, 35.806, 107.898, 0]
  MoveL 336 to (0, -242.61, -60.35) mm, rotated rx -90 ry 0 rz -90 deg; joints [-17.921, -100.434, -115.263, 35.697, 107.921, 0]
  MoveL 337 to (0, -242.85, -59.38) mm, rotated rx -90 ry 0 rz -90 deg; joints [-17.943, -100.387, -115.201, 35.588, 107.943, 0]
  MoveL 338 to (0, -243.08, -58.41) mm, rotated rx -90 ry 0 rz -90 deg; joints [-17.966, -100.341, -115.139, 35.48, 107.966, 0]
  MoveL 339 to (0, -243.31, -57.44) mm, rotated rx -90 ry 0 rz -90 deg; joints [-17.988, -100.294, -115.077, 35.371, 107.988, 0]
  MoveL 340 to (0, -243.54, -56.46) mm, rotated rx -90 ry 0 rz -90 deg; joints [-18.009, -100.247, -115.015, 35.262, 108.009, 0]
  MoveL 341 to (0, -243.76, -55.49) mm, rotated rx -90 ry 0 rz -90 deg; joints [-18.03, -100.201, -114.953, 35.154, 108.03, 0]
  MoveL 342 to (0, -243.98, -54.52) mm, rotated rx -90 ry 0 rz -90 deg; joints [-18.051, -100.154, -114.891, 35.045, 108.051, 0]
  MoveL 343 to (0, -244.2, -53.54) mm, rotated rx -90 ry 0 rz -90 deg; joints [-18.072, -100.107, -114.829, 34.936, 108.072, 0]
  MoveL 344 to (0, -244.41, -52.56) mm, rotated rx -90 ry 0 rz -90 deg; joints [-18.092, -100.06, -114.767, 34.828, 108.092, 0]
  MoveL 345 to (0, -244.62, -51.59) mm, rotated rx -90 ry 0 rz -90 deg; joints [-18.111, -100.014, -114.705, 34.719, 108.111, 0]
  MoveL 346 to (0, -244.82, -50.61) mm, rotated rx -90 ry 0 rz -90 deg; joints [-18.131, -99.967, -114.644, 34.61, 108.131, 0]
  MoveL 347 to (0, -245.02, -49.63) mm, rotated rx -90 ry 0 rz -90 deg; joints [-18.149, -99.92, -114.582, 34.502, 108.15, 0]
  MoveL 348 to (0, -245.22, -48.65) mm, rotated rx -90 ry 0 rz -90 deg; joints [-18.168, -99.873, -114.52, 34.393, 108.168, 0]
  MoveL 349 to (0, -245.41, -47.67) mm, rotated rx -90 ry 0 rz -90 deg; joints [-18.186, -99.826, -114.459, 34.284, 108.186, 0]
  MoveL 350 to (0, -245.6, -46.69) mm, rotated rx -90 ry 0 rz -90 deg; joints [-18.204, -99.778, -114.397, 34.176, 108.204, 0]
  MoveL 351 to (0, -245.79, -45.71) mm, rotated rx -90 ry 0 rz -90 deg; joints [-18.221, -99.731, -114.336, 34.067, 108.221, 0]
  MoveL 352 to (0, -245.97, -44.72) mm, rotated rx -90 ry 0 rz -90 deg; joints [-18.238, -99.684, -114.274, 33.959, 108.239, 0]
  MoveL 353 to (0, -246.14, -43.74) mm, rotated rx -90 ry 0 rz -90 deg; joints [-18.255, -99.637, -114.213, 33.85, 108.255, 0]
  MoveL 354 to (0, -246.32, -42.76) mm, rotated rx -90 ry 0 rz -90 deg; joints [-18.271, -99.59, -114.152, 33.741, 108.271, 0]
  MoveL 355 to (0, -246.49, -41.77) mm, rotated rx -90 ry 0 rz -90 deg; joints [-18.287, -99.542, -114.091, 33.633, 108.287, 0]
  MoveL 356 to (0, -246.65, -40.79) mm, rotated rx -90 ry 0 rz -90 deg; joints [-18.303, -99.495, -114.029, 33.524, 108.303, 0]
  MoveL 357 to (0, -246.81, -39.8) mm, rotated rx -90 ry 0 rz -90 deg; joints [-18.318, -99.447, -113.968, 33.416, 108.318, 0]
  MoveL 358 to (0, -246.97, -38.81) mm, rotated rx -90 ry 0 rz -90 deg; joints [-18.333, -99.4, -113.907, 33.307, 108.333, 0]
  MoveL 359 to (0, -247.12, -37.83) mm, rotated rx -90 ry 0 rz -90 deg; joints [-18.347, -99.353, -113.846, 33.199, 108.347, 0]
  MoveL 360 to (0, -247.27, -36.84) mm, rotated rx -90 ry 0 rz -90 deg; joints [-18.361, -99.305, -113.785, 33.09, 108.361, 0]
  MoveL 361 to (0, -247.42, -35.85) mm, rotated rx -90 ry 0 rz -90 deg; joints [-18.375, -99.257, -113.725, 32.982, 108.375, 0]
  MoveL 362 to (0, -247.56, -34.86) mm, rotated rx -90 ry 0 rz -90 deg; joints [-18.388, -99.21, -113.664, 32.873, 108.388, 0]
  MoveL 363 to (0, -247.7, -33.87) mm, rotated rx -90 ry 0 rz -90 deg; joints [-18.401, -99.162, -113.603, 32.765, 108.401, 0]
  MoveL 364 to (0, -247.83, -32.88) mm, rotated rx -90 ry 0 rz -90 deg; joints [-18.414, -99.114, -113.542, 32.657, 108.414, 0]
  MoveL 365 to (0, -247.96, -31.89) mm, rotated rx -90 ry 0 rz -90 deg; joints [-18.426, -99.067, -113.482, 32.548, 108.426, 0]
  MoveL 366 to (0, -248.08, -30.9) mm, rotated rx -90 ry 0 rz -90 deg; joints [-18.438, -99.019, -113.421, 32.44, 108.438, 0]
  MoveL 367 to (0, -248.2, -29.91) mm, rotated rx -90 ry 0 rz -90 deg; joints [-18.449, -98.971, -113.361, 32.332, 108.449, 0]
  MoveL 368 to (0, -248.32, -28.91) mm, rotated rx -90 ry 0 rz -90 deg; joints [-18.46, -98.923, -113.3, 32.224, 108.46, 0]
  MoveL 369 to (0, -248.44, -27.92) mm, rotated rx -90 ry 0 rz -90 deg; joints [-18.471, -98.875, -113.24, 32.115, 108.471, 0]
  MoveL 370 to (0, -248.55, -26.93) mm, rotated rx -90 ry 0 rz -90 deg; joints [-18.481, -98.827, -113.18, 32.007, 108.481, 0]
  MoveL 371 to (0, -248.65, -25.93) mm, rotated rx -90 ry 0 rz -90 deg; joints [-18.491, -98.779, -113.12, 31.899, 108.491, 0]
  MoveL 372 to (0, -248.75, -24.94) mm, rotated rx -90 ry 0 rz -90 deg; joints [-18.501, -98.731, -113.06, 31.791, 108.501, 0]
  MoveL 373 to (0, -248.85, -23.94) mm, rotated rx -90 ry 0 rz -90 deg; joints [-18.51, -98.683, -113, 31.683, 108.51, 0]
  MoveL 374 to (0, -248.94, -22.95) mm, rotated rx -90 ry 0 rz -90 deg; joints [-18.519, -98.635, -112.94, 31.575, 108.519, 0]
  MoveL 375 to (0, -249.03, -21.95) mm, rotated rx -90 ry 0 rz -90 deg; joints [-18.527, -98.587, -112.88, 31.467, 108.527, 0]
  MoveL 376 to (0, -249.12, -20.96) mm, rotated rx -90 ry 0 rz -90 deg; joints [-18.535, -98.539, -112.82, 31.359, 108.535, 0]
  MoveL 377 to (0, -249.2, -19.96) mm, rotated rx -90 ry 0 rz -90 deg; joints [-18.543, -98.49, -112.76, 31.251, 108.543, 0]
  MoveL 378 to (0, -249.28, -18.97) mm, rotated rx -90 ry 0 rz -90 deg; joints [-18.55, -98.442, -112.701, 31.143, 108.55, 0]
  MoveL 379 to (0, -249.35, -17.97) mm, rotated rx -90 ry 0 rz -90 deg; joints [-18.557, -98.394, -112.641, 31.035, 108.557, 0]
  MoveL 380 to (0, -249.42, -16.97) mm, rotated rx -90 ry 0 rz -90 deg; joints [-18.564, -98.346, -112.582, 30.927, 108.564, 0]
  MoveL 381 to (0, -249.49, -15.98) mm, rotated rx -90 ry 0 rz -90 deg; joints [-18.57, -98.297, -112.522, 30.82, 108.57, 0]
  MoveL 382 to (0, -249.55, -14.98) mm, rotated rx -90 ry 0 rz -90 deg; joints [-18.576, -98.249, -112.463, 30.712, 108.576, 0]
  MoveL 383 to (0, -249.61, -13.98) mm, rotated rx -90 ry 0 rz -90 deg; joints [-18.581, -98.2, -112.404, 30.604, 108.581, 0]
  MoveL 384 to (0, -249.66, -12.98) mm, rotated rx -90 ry 0 rz -90 deg; joints [-18.586, -98.152, -112.345, 30.497, 108.586, 0]
  MoveL 385 to (0, -249.71, -11.99) mm, rotated rx -90 ry 0 rz -90 deg; joints [-18.591, -98.103, -112.286, 30.389, 108.591, 0]
  MoveL 386 to (0, -249.76, -10.99) mm, rotated rx -90 ry 0 rz -90 deg; joints [-18.595, -98.055, -112.227, 30.281, 108.595, 0]
  MoveL 387 to (0, -249.8, -9.99) mm, rotated rx -90 ry 0 rz -90 deg; joints [-18.599, -98.006, -112.168, 30.174, 108.599, 0]
  MoveL 388 to (0, -249.84, -8.99) mm, rotated rx -90 ry 0 rz -90 deg; joints [-18.602, -97.958, -112.109, 30.067, 108.603, 0]
  MoveL 389 to (0, -249.87, -7.99) mm, rotated rx -90 ry 0 rz -90 deg; joints [-18.606, -97.909, -112.05, 29.959, 108.606, 0]
  MoveL 390 to (0, -249.9, -6.99) mm, rotated rx -90 ry 0 rz -90 deg; joints [-18.608, -97.86, -111.991, 29.852, 108.609, 0]
  MoveL 391 to (0, -249.93, -5.99) mm, rotated rx -90 ry 0 rz -90 deg; joints [-18.611, -97.812, -111.933, 29.745, 108.611, 0]
  MoveL 392 to (0, -249.95, -5) mm, rotated rx -90 ry 0 rz -90 deg; joints [-18.613, -97.763, -111.874, 29.638, 108.613, 0]
  MoveL 393 to (0, -249.97, -4) mm, rotated rx -90 ry 0 rz -90 deg; joints [-18.615, -97.714, -111.816, 29.53, 108.615, 0]
  MoveL 394 to (0, -249.98, -3) mm, rotated rx -90 ry 0 rz -90 deg; joints [-18.616, -97.666, -111.758, 29.423, 108.616, 0]
  MoveL 395 to (0, -249.99, -2) mm, rotated rx -90 ry 0 rz -90 deg; joints [-18.617, -97.617, -111.7, 29.316, 108.617, 0]
  MoveL 396 to (0, -250, -1) mm, rotated rx -90 ry 0 rz -90 deg; joints [-18.617, -97.568, -111.642, 29.209, 108.618, 0]
  MoveL 397 to (0, -250, 0) mm, rotated rx -90 ry 0 rz -90 deg; joints [-18.618, -97.519, -111.584, 29.103, 108.618, 0]
  MoveL 398 to (0, -250, 1) mm, rotated rx -90 ry 0 rz -90 deg; joints [-18.617, -97.47, -111.526, 28.996, 108.618, 0]
  MoveL 399 to (0, -249.99, 2) mm, rotated rx -90 ry 0 rz -90 deg; joints [-18.617, -97.421, -111.468, 28.889, 108.617, 0]
  MoveL 400 to (0, -249.98, 3) mm, rotated rx -90 ry 0 rz -90 deg; joints [-18.616, -97.372, -111.41, 28.782, 108.616, 0]
  MoveL 401 to (0, -249.97, 4) mm, rotated rx -90 ry 0 rz -90 deg; joints [-18.615, -97.323, -111.353, 28.676, 108.615, 0]
  MoveL 402 to (0, -249.95, 5) mm, rotated rx -90 ry 0 rz -90 deg; joints [-18.613, -97.274, -111.295, 28.569, 108.613, 0]
  MoveL 403 to (0, -249.93, 5.99) mm, rotated rx -90 ry 0 rz -90 deg; joints [-18.611, -97.225, -111.238, 28.463, 108.611, 0]
  MoveL 404 to (0, -249.9, 6.99) mm, rotated rx -90 ry 0 rz -90 deg; joints [-18.608, -97.176, -111.18, 28.356, 108.609, 0]
  MoveL 405 to (0, -249.87, 7.99) mm, rotated rx -90 ry 0 rz -90 deg; joints [-18.606, -97.127, -111.123, 28.25, 108.606, 0]
  MoveL 406 to (0, -249.84, 8.99) mm, rotated rx -90 ry 0 rz -90 deg; joints [-18.602, -97.078, -111.066, 28.144, 108.603, 0]
  MoveL 407 to (0, -249.8, 9.99) mm, rotated rx -90 ry 0 rz -90 deg; joints [-18.599, -97.029, -111.009, 28.038, 108.599, 0]
  MoveL 408 to (0, -249.76, 10.99) mm, rotated rx -90 ry 0 rz -90 deg; joints [-18.595, -96.98, -110.952, 27.932, 108.595, 0]
  MoveL 409 to (0, -249.71, 11.99) mm, rotated rx -90 ry 0 rz -90 deg; joints [-18.591, -96.93, -110.895, 27.826, 108.591, 0]
  MoveL 410 to (0, -249.66, 12.98) mm, rotated rx -90 ry 0 rz -90 deg; joints [-18.586, -96.881, -110.838, 27.72, 108.586, 0]
  MoveL 411 to (0, -249.61, 13.98) mm, rotated rx -90 ry 0 rz -90 deg; joints [-18.581, -96.832, -110.782, 27.614, 108.581, 0]
  MoveL 412 to (0, -249.55, 14.98) mm, rotated rx -90 ry 0 rz -90 deg; joints [-18.576, -96.783, -110.725, 27.508, 108.576, 0]
  MoveL 413 to (0, -249.49, 15.98) mm, rotated rx -90 ry 0 rz -90 deg; joints [-18.57, -96.733, -110.669, 27.402, 108.57, 0]
  MoveL 414 to (0, -249.42, 16.97) mm, rotated rx -90 ry 0 rz -90 deg; joints [-18.564, -96.684, -110.612, 27.297, 108.564, 0]
  MoveL 415 to (0, -249.35, 17.97) mm, rotated rx -90 ry 0 rz -90 deg; joints [-18.557, -96.635, -110.556, 27.191, 108.557, 0]
  MoveL 416 to (0, -249.28, 18.97) mm, rotated rx -90 ry 0 rz -90 deg; joints [-18.55, -96.585, -110.5, 27.086, 108.55, 0]
  MoveL 417 to (0, -249.2, 19.96) mm, rotated rx -90 ry 0 rz -90 deg; joints [-18.543, -96.536, -110.444, 26.98, 108.543, 0]
  MoveL 418 to (0, -249.12, 20.96) mm, rotated rx -90 ry 0 rz -90 deg; joints [-18.535, -96.487, -110.388, 26.875, 108.535, 0]
  MoveL 419 to (0, -249.03, 21.95) mm, rotated rx -90 ry 0 rz -90 deg; joints [-18.527, -96.437, -110.333, 26.77, 108.527, 0]
  MoveL 420 to (0, -248.94, 22.95) mm, rotated rx -90 ry 0 rz -90 deg; joints [-18.519, -96.388, -110.277, 26.665, 108.519, 0]
  MoveL 421 to (0, -248.85, 23.94) mm, rotated rx -90 ry 0 rz -90 deg; joints [-18.51, -96.338, -110.221, 26.56, 108.51, 0]
  MoveL 422 to (0, -248.75, 24.94) mm, rotated rx -90 ry 0 rz -90 deg; joints [-18.501, -96.289, -110.166, 26.455, 108.501, 0]
  MoveL 423 to (0, -248.65, 25.93) mm, rotated rx -90 ry 0 rz -90 deg; joints [-18.491, -96.239, -110.111, 26.35, 108.491, 0]
  MoveL 424 to (0, -248.55, 26.93) mm, rotated rx -90 ry 0 rz -90 deg; joints [-18.481, -96.19, -110.055, 26.245, 108.481, 0]
  MoveL 425 to (0, -248.44, 27.92) mm, rotated rx -90 ry 0 rz -90 deg; joints [-18.471, -96.14, -110, 26.141, 108.471, 0]
  MoveL 426 to (0, -248.32, 28.91) mm, rotated rx -90 ry 0 rz -90 deg; joints [-18.46, -96.091, -109.945, 26.036, 108.46, 0]
  MoveL 427 to (0, -248.2, 29.91) mm, rotated rx -90 ry 0 rz -90 deg; joints [-18.449, -96.041, -109.89, 25.932, 108.449, 0]
  MoveL 428 to (0, -248.08, 30.9) mm, rotated rx -90 ry 0 rz -90 deg; joints [-18.438, -95.992, -109.836, 25.827, 108.438, 0]
  MoveL 429 to (0, -247.96, 31.89) mm, rotated rx -90 ry 0 rz -90 deg; joints [-18.426, -95.942, -109.781, 25.723, 108.426, 0]
  MoveL 430 to (0, -247.83, 32.88) mm, rotated rx -90 ry 0 rz -90 deg; joints [-18.414, -95.892, -109.726, 25.619, 108.414, 0]
  MoveL 431 to (0, -247.7, 33.87) mm, rotated rx -90 ry 0 rz -90 deg; joints [-18.401, -95.843, -109.672, 25.515, 108.401, 0]
  MoveL 432 to (0, -247.56, 34.86) mm, rotated rx -90 ry 0 rz -90 deg; joints [-18.388, -95.793, -109.618, 25.411, 108.388, 0]
  MoveL 433 to (0, -247.42, 35.85) mm, rotated rx -90 ry 0 rz -90 deg; joints [-18.375, -95.743, -109.564, 25.307, 108.375, 0]
  MoveL 434 to (0, -247.27, 36.84) mm, rotated rx -90 ry 0 rz -90 deg; joints [-18.361, -95.694, -109.51, 25.203, 108.361, 0]
  MoveL 435 to (0, -247.12, 37.83) mm, rotated rx -90 ry 0 rz -90 deg; joints [-18.347, -95.644, -109.456, 25.1, 108.347, 0]
  MoveL 436 to (0, -246.97, 38.81) mm, rotated rx -90 ry 0 rz -90 deg; joints [-18.333, -95.594, -109.402, 24.996, 108.333, 0]
  MoveL 437 to (0, -246.81, 39.8) mm, rotated rx -90 ry 0 rz -90 deg; joints [-18.318, -95.544, -109.348, 24.893, 108.318, 0]
  MoveL 438 to (0, -246.65, 40.79) mm, rotated rx -90 ry 0 rz -90 deg; joints [-18.303, -95.495, -109.295, 24.789, 108.303, 0]
  MoveL 439 to (0, -246.49, 41.77) mm, rotated rx -90 ry 0 rz -90 deg; joints [-18.287, -95.445, -109.241, 24.686, 108.287, 0]
  MoveL 440 to (0, -246.32, 42.76) mm, rotated rx -90 ry 0 rz -90 deg; joints [-18.271, -95.395, -109.188, 24.583, 108.271, 0]
  MoveL 441 to (0, -246.14, 43.74) mm, rotated rx -90 ry 0 rz -90 deg; joints [-18.255, -95.345, -109.135, 24.48, 108.255, 0]
  MoveL 442 to (0, -245.97, 44.72) mm, rotated rx -90 ry 0 rz -90 deg; joints [-18.238, -95.295, -109.081, 24.377, 108.239, 0]
  MoveL 443 to (0, -245.79, 45.71) mm, rotated rx -90 ry 0 rz -90 deg; joints [-18.221, -95.246, -109.029, 24.274, 108.221, 0]
  MoveL 444 to (0, -245.6, 46.69) mm, rotated rx -90 ry 0 rz -90 deg; joints [-18.204, -95.196, -108.976, 24.172, 108.204, 0]
  MoveL 445 to (0, -245.41, 47.67) mm, rotated rx -90 ry 0 rz -90 deg; joints [-18.186, -95.146, -108.923, 24.069, 108.186, 0]
  MoveL 446 to (0, -245.22, 48.65) mm, rotated rx -90 ry 0 rz -90 deg; joints [-18.168, -95.096, -108.87, 23.967, 108.168, 0]
  MoveL 447 to (0, -245.02, 49.63) mm, rotated rx -90 ry 0 rz -90 deg; joints [-18.149, -95.046, -108.818, 23.864, 108.15, 0]
  MoveL 448 to (0, -244.82, 50.61) mm, rotated rx -90 ry 0 rz -90 deg; joints [-18.131, -94.996, -108.766, 23.762, 108.131, 0]
  MoveL 449 to (0, -244.62, 51.59) mm, rotated rx -90 ry 0 rz -90 deg; joints [-18.111, -94.946, -108.714, 23.66, 108.111, 0]
  MoveL 450 to (0, -244.41, 52.56) mm, rotated rx -90 ry 0 rz -90 deg; joints [-18.092, -94.897, -108.662, 23.558, 108.092, 0]
  MoveL 451 to (0, -244.2, 53.54) mm, rotated rx -90 ry 0 rz -90 deg; joints [-18.072, -94.847, -108.61, 23.456, 108.072, 0]
  MoveL 452 to (0, -243.98, 54.52) mm, rotated rx -90 ry 0 rz -90 deg; joints [-18.051, -94.797, -108.558, 23.355, 108.051, 0]
  MoveL 453 to (0, -243.76, 55.49) mm, rotated rx -90 ry 0 rz -90 deg; joints [-18.03, -94.747, -108.506, 23.253, 108.03, 0]
  MoveL 454 to (0, -243.54, 56.46) mm, rotated rx -90 ry 0 rz -90 deg; joints [-18.009, -94.697, -108.455, 23.152, 108.009, 0]
  MoveL 455 to (0, -243.31, 57.44) mm, rotated rx -90 ry 0 rz -90 deg; joints [-17.988, -94.647, -108.403, 23.05, 107.988, 0]
  MoveL 456 to (0, -243.08, 58.41) mm, rotated rx -90 ry 0 rz -90 deg; joints [-17.966, -94.597, -108.352, 22.949, 107.966, 0]
  MoveL 457 to (0, -242.85, 59.38) mm, rotated rx -90 ry 0 rz -90 deg; joints [-17.943, -94.547, -108.301, 22.848, 107.943, 0]
  MoveL 458 to (0, -242.61, 60.35) mm, rotated rx -90 ry 0 rz -90 deg; joints [-17.921, -94.497, -108.25, 22.747, 107.921, 0]
  MoveL 459 to (0, -242.36, 61.32) mm, rotated rx -90 ry 0 rz -90 deg; joints [-17.898, -94.447, -108.199, 22.646, 107.898, 0]
  MoveL 460 to (0, -242.12, 62.29) mm, rotated rx -90 ry 0 rz -90 deg; joints [-17.874, -94.397, -108.148, 22.545, 107.874, 0]
  MoveL 461 to (0, -241.87, 63.26) mm, rotated rx -90 ry 0 rz -90 deg; joints [-17.85, -94.347, -108.098, 22.445, 107.85, 0]
  MoveL 462 to (0, -241.61, 64.22) mm, rotated rx -90 ry 0 rz -90 deg; joints [-17.826, -94.297, -108.047, 22.344, 107.826, 0]
  MoveL 463 to (0, -241.35, 65.19) mm, rotated rx -90 ry 0 rz -90 deg; joints [-17.802, -94.247, -107.997, 22.244, 107.802, 0]
  MoveL 464 to (0, -241.09, 66.15) mm, rotated rx -90 ry 0 rz -90 deg; joints [-17.777, -94.197, -107.947, 22.144, 107.777, 0]
  MoveL 465 to (0, -240.82, 67.11) mm, rotated rx -90 ry 0 rz -90 deg; joints [-17.751, -94.147, -107.897, 22.044, 107.751, 0]
  MoveL 466 to (0, -240.55, 68.08) mm, rotated rx -90 ry 0 rz -90 deg; joints [-17.726, -94.097, -107.847, 21.944, 107.726, 0]
  MoveL 467 to (0, -240.28, 69.04) mm, rotated rx -90 ry 0 rz -90 deg; joints [-17.7, -94.047, -107.797, 21.844, 107.7, 0]
  MoveL 468 to (0, -240, 70) mm, rotated rx -90 ry 0 rz -90 deg; joints [-17.673, -93.997, -107.748, 21.745, 107.673, 0]
  MoveL 469 to (0, -239.72, 70.96) mm, rotated rx -90 ry 0 rz -90 deg; joints [-17.646, -93.947, -107.698, 21.645, 107.646, 0]
  MoveL 470 to (0, -239.43, 71.91) mm, rotated rx -90 ry 0 rz -90 deg; joints [-17.619, -93.897, -107.649, 21.546, 107.619, 0]
  MoveL 471 to (0, -239.14, 72.87) mm, rotated rx -90 ry 0 rz -90 deg; joints [-17.591, -93.847, -107.6, 21.447, 107.592, 0]
  MoveL 472 to (0, -238.85, 73.83) mm, rotated rx -90 ry 0 rz -90 deg; joints [-17.564, -93.797, -107.551, 21.348, 107.564, 0]
  MoveL 473 to (0, -238.55, 74.78) mm, rotated rx -90 ry 0 rz -90 deg; joints [-17.535, -93.747, -107.502, 21.249, 107.535, 0]
  MoveL 474 to (0, -238.25, 75.73) mm, rotated rx -90 ry 0 rz -90 deg; joints [-17.506, -93.697, -107.453, 21.15, 107.507, 0]
  MoveL 475 to (0, -237.95, 76.68) mm, rotated rx -90 ry 0 rz -90 deg; joints [-17.477, -93.647, -107.405, 21.051, 107.477, 0]
  MoveL 476 to (0, -237.64, 77.63) mm, rotated rx -90 ry 0 rz -90 deg; joints [-17.448, -93.597, -107.356, 20.953, 107.448, 0]
  MoveL 477 to (0, -237.33, 78.58) mm, rotated rx -90 ry 0 rz -90 deg; joints [-17.418, -93.547, -107.308, 20.855, 107.418, 0]
  MoveL 478 to (0, -237.01, 79.53) mm, rotated rx -90 ry 0 rz -90 deg; joints [-17.388, -93.496, -107.26, 20.756, 107.388, 0]
  MoveL 479 to (0, -236.69, 80.48) mm, rotated rx -90 ry 0 rz -90 deg; joints [-17.357, -93.446, -107.212, 20.658, 107.357, 0]
  MoveL 480 to (0, -236.37, 81.42) mm, rotated rx -90 ry 0 rz -90 deg; joints [-17.326, -93.396, -107.164, 20.561, 107.326, 0]
  MoveL 481 to (0, -236.04, 82.37) mm, rotated rx -90 ry 0 rz -90 deg; joints [-17.295, -93.346, -107.116, 20.463, 107.295, 0]
  MoveL 482 to (0, -235.71, 83.31) mm, rotated rx -90 ry 0 rz -90 deg; joints [-17.263, -93.296, -107.069, 20.365, 107.263, 0]
  MoveL 483 to (0, -235.38, 84.25) mm, rotated rx -90 ry 0 rz -90 deg; joints [-17.231, -93.246, -107.022, 20.268, 107.231, 0]
  MoveL 484 to (0, -235.04, 85.19) mm, rotated rx -90 ry 0 rz -90 deg; joints [-17.199, -93.196, -106.974, 20.171, 107.199, 0]
  MoveL 485 to (0, -234.69, 86.13) mm, rotated rx -90 ry 0 rz -90 deg; joints [-17.166, -93.146, -106.927, 20.073, 107.166, 0]
  MoveL 486 to (0, -234.35, 87.07) mm, rotated rx -90 ry 0 rz -90 deg; joints [-17.133, -93.096, -106.88, 19.977, 107.133, 0]
  MoveL 487 to (0, -234, 88) mm, rotated rx -90 ry 0 rz -90 deg; joints [-17.099, -93.046, -106.834, 19.88, 107.099, 0]
  MoveL 488 to (0, -233.64, 88.94) mm, rotated rx -90 ry 0 rz -90 deg; joints [-17.065, -92.996, -106.787, 19.783, 107.065, 0]
  MoveL 489 to (0, -233.29, 89.87) mm, rotated rx -90 ry 0 rz -90 deg; joints [-17.031, -92.946, -106.741, 19.687, 107.031, 0]
  MoveL 490 to (0, -232.93, 90.8) mm, rotated rx -90 ry 0 rz -90 deg; joints [-16.996, -92.896, -106.694, 19.59, 106.996, 0]
  MoveL 491 to (0, -232.56, 91.73) mm, rotated rx -90 ry 0 rz -90 deg; joints [-16.961, -92.846, -106.648, 19.494, 106.961, 0]
  MoveL 492 to (0, -232.19, 92.66) mm, rotated rx -90 ry 0 rz -90 deg; joints [-16.925, -92.796, -106.602, 19.398, 106.925, 0]
  MoveL 493 to (0, -231.82, 93.59) mm, rotated rx -90 ry 0 rz -90 deg; joints [-16.889, -92.746, -106.556, 19.302, 106.889, 0]
  MoveL 494 to (0, -231.44, 94.52) mm, rotated rx -90 ry 0 rz -90 deg; joints [-16.853, -92.696, -106.511, 19.207, 106.853, 0]
  MoveL 495 to (0, -231.07, 95.44) mm, rotated rx -90 ry 0 rz -90 deg; joints [-16.816, -92.646, -106.465, 19.111, 106.816, 0]
  MoveL 496 to (0, -230.68, 96.36) mm, rotated rx -90 ry 0 rz -90 deg; joints [-16.779, -92.596, -106.42, 19.016, 106.779, 0]
  MoveL 497 to (0, -230.3, 97.28) mm, rotated rx -90 ry 0 rz -90 deg; joints [-16.742, -92.546, -106.375, 18.921, 106.742, 0]
  MoveL 498 to (0, -229.9, 98.2) mm, rotated rx -90 ry 0 rz -90 deg; joints [-16.704, -92.496, -106.33, 18.826, 106.704, 0]
  MoveL 499 to (0, -229.51, 99.12) mm, rotated rx -90 ry 0 rz -90 deg; joints [-16.666, -92.446, -106.285, 18.731, 106.666, 0]
  MoveL 500 to (0, -229.11, 100.04) mm, rotated rx -90 ry 0 rz -90 deg; joints [-16.628, -92.396, -106.24, 18.636, 106.628, 0]
  MoveL 501 to (0, -228.71, 100.95) mm, rotated rx -90 ry 0 rz -90 deg; joints [-16.589, -92.346, -106.195, 18.542, 106.589, 0]
  MoveL 502 to (0, -228.31, 101.87) mm, rotated rx -90 ry 0 rz -90 deg; joints [-16.549, -92.297, -106.151, 18.448, 106.549, 0]
  MoveL 503 to (0, -227.9, 102.78) mm, rotated rx -90 ry 0 rz -90 deg; joints [-16.51, -92.247, -106.107, 18.353, 106.51, 0]
  MoveL 504 to (0, -227.48, 103.69) mm, rotated rx -90 ry 0 rz -90 deg; joints [-16.47, -92.197, -106.063, 18.26, 106.47, 0]
  MoveL 505 to (0, -227.07, 104.6) mm, rotated rx -90 ry 0 rz -90 deg; joints [-16.429, -92.147, -106.019, 18.166, 106.429, 0]
  MoveL 506 to (0, -226.65, 105.5) mm, rotated rx -90 ry 0 rz -90 deg; joints [-16.388, -92.097, -105.975, 18.072, 106.388, 0]
  MoveL 507 to (0, -226.22, 106.41) mm, rotated rx -90 ry 0 rz -90 deg; joints [-16.347, -92.047, -105.932, 17.979, 106.347, 0]
  MoveL 508 to (0, -225.8, 107.31) mm, rotated rx -90 ry 0 rz -90 deg; joints [-16.306, -91.997, -105.888, 17.886, 106.306, 0]
  MoveL 509 to (0, -225.37, 108.21) mm, rotated rx -90 ry 0 rz -90 deg; joints [-16.264, -91.947, -105.845, 17.792, 106.264, 0]
  MoveL 510 to (0, -224.93, 109.11) mm, rotated rx -90 ry 0 rz -90 deg; joints [-16.221, -91.898, -105.802, 17.7, 106.222, 0]
  MoveL 511 to (0, -224.49, 110.01) mm, rotated rx -90 ry 0 rz -90 deg; joints [-16.179, -91.848, -105.759, 17.607, 106.179, 0]
  MoveL 512 to (0, -224.05, 110.91) mm, rotated rx -90 ry 0 rz -90 deg; joints [-16.136, -91.798, -105.716, 17.514, 106.136, 0]
  MoveL 513 to (0, -223.61, 111.8) mm, rotated rx -90 ry 0 rz -90 deg; joints [-16.092, -91.748, -105.674, 17.422, 106.092, 0]
  MoveL 514 to (0, -223.16, 112.7) mm, rotated rx -90 ry 0 rz -90 deg; joints [-16.048, -91.698, -105.631, 17.33, 106.049, 0]
  MoveL 515 to (0, -222.71, 113.59) mm, rotated rx -90 ry 0 rz -90 deg; joints [-16.004, -91.649, -105.589, 17.238, 106.004, 0]
  MoveL 516 to (0, -222.25, 114.48) mm, rotated rx -90 ry 0 rz -90 deg; joints [-15.96, -91.599, -105.547, 17.146, 105.96, 0]
  MoveL 517 to (0, -221.79, 115.36) mm, rotated rx -90 ry 0 rz -90 deg; joints [-15.915, -91.549, -105.505, 17.055, 105.915, 0]
  MoveL 518 to (0, -221.33, 116.25) mm, rotated rx -90 ry 0 rz -90 deg; joints [-15.869, -91.5, -105.464, 16.963, 105.869, 0]
  MoveL 519 to (0, -220.86, 117.13) mm, rotated rx -90 ry 0 rz -90 deg; joints [-15.824, -91.45, -105.422, 16.872, 105.824, 0]
  MoveL 520 to (0, -220.39, 118.01) mm, rotated rx -90 ry 0 rz -90 deg; joints [-15.778, -91.4, -105.381, 16.781, 105.778, 0]
  MoveL 521 to (0, -219.92, 118.89) mm, rotated rx -90 ry 0 rz -90 deg; joints [-15.731, -91.351, -105.34, 16.69, 105.731, 0]
  MoveL 522 to (0, -219.44, 119.77) mm, rotated rx -90 ry 0 rz -90 deg; joints [-15.684, -91.301, -105.299, 16.6, 105.684, 0]
  MoveL 523 to (0, -218.96, 120.65) mm, rotated rx -90 ry 0 rz -90 deg; joints [-15.637, -91.251, -105.258, 16.509, 105.637, 0]
  MoveL 524 to (0, -218.48, 121.52) mm, rotated rx -90 ry 0 rz -90 deg; joints [-15.589, -91.202, -105.217, 16.419, 105.589, 0]
  MoveL 525 to (0, -217.99, 122.39) mm, rotated rx -90 ry 0 rz -90 deg; joints [-15.541, -91.152, -105.177, 16.329, 105.542, 0]
  MoveL 526 to (0, -217.5, 123.27) mm, rotated rx -90 ry 0 rz -90 deg; joints [-15.493, -91.103, -105.136, 16.239, 105.493, 0]
  MoveL 527 to (0, -217, 124.13) mm, rotated rx -90 ry 0 rz -90 deg; joints [-15.444, -91.053, -105.096, 16.149, 105.444, 0]
  MoveL 528 to (0, -216.51, 125) mm, rotated rx -90 ry 0 rz -90 deg; joints [-15.395, -91.004, -105.056, 16.06, 105.395, 0]
  MoveL 529 to (0, -216.01, 125.86) mm, rotated rx -90 ry 0 rz -90 deg; joints [-15.346, -90.954, -105.016, 15.971, 105.346, 0]
  MoveL 530 to (0, -215.5, 126.73) mm, rotated rx -90 ry 0 rz -90 deg; joints [-15.296, -90.905, -104.977, 15.882, 105.296, 0]
  MoveL 531 to (0, -214.99, 127.59) mm, rotated rx -90 ry 0 rz -90 deg; joints [-15.246, -90.855, -104.937, 15.793, 105.246, 0]
  MoveL 532 to (0, -214.48, 128.45) mm, rotated rx -90 ry 0 rz -90 deg; joints [-15.195, -90.806, -104.898, 15.704, 105.195, 0]
  MoveL 533 to (0, -213.97, 129.3) mm, rotated rx -90 ry 0 rz -90 deg; joints [-15.144, -90.757, -104.859, 15.616, 105.144, 0]
  MoveL 534 to (0, -213.45, 130.16) mm, rotated rx -90 ry 0 rz -90 deg; joints [-15.093, -90.707, -104.82, 15.528, 105.093, 0]
  MoveL 535 to (0, -212.92, 131.01) mm, rotated rx -90 ry 0 rz -90 deg; joints [-15.041, -90.658, -104.782, 15.44, 105.041, 0]
  MoveL 536 to (0, -212.4, 131.86) mm, rotated rx -90 ry 0 rz -90 deg; joints [-14.989, -90.609, -104.743, 15.352, 104.989, 0]
  MoveL 537 to (0, -211.87, 132.71) mm, rotated rx -90 ry 0 rz -90 deg; joints [-14.936, -90.559, -104.705, 15.264, 104.936, 0]
  MoveL 538 to (0, -211.34, 133.55) mm, rotated rx -90 ry 0 rz -90 deg; joints [-14.883, -90.51, -104.667, 15.177, 104.883, 0]
  MoveL 539 to (0, -210.8, 134.4) mm, rotated rx -90 ry 0 rz -90 deg; joints [-14.83, -90.461, -104.629, 15.09, 104.83, 0]
  MoveL 540 to (0, -210.26, 135.24) mm, rotated rx -90 ry 0 rz -90 deg; joints [-14.776, -90.412, -104.591, 15.003, 104.776, 0]
  MoveL 541 to (0, -209.72, 136.08) mm, rotated rx -90 ry 0 rz -90 deg; joints [-14.722, -90.363, -104.553, 14.916, 104.722, 0]
  MoveL 542 to (0, -209.18, 136.91) mm, rotated rx -90 ry 0 rz -90 deg; joints [-14.668, -90.314, -104.516, 14.829, 104.668, 0]
  MoveL 543 to (0, -208.63, 137.75) mm, rotated rx -90 ry 0 rz -90 deg; joints [-14.613, -90.264, -104.479, 14.743, 104.613, 0]
  MoveL 544 to (0, -208.08, 138.58) mm, rotated rx -90 ry 0 rz -90 deg; joints [-14.558, -90.215, -104.442, 14.657, 104.558, 0]
  MoveL 545 to (0, -207.52, 139.41) mm, rotated rx -90 ry 0 rz -90 deg; joints [-14.503, -90.166, -104.405, 14.571, 104.503, 0]
  MoveL 546 to (0, -206.96, 140.24) mm, rotated rx -90 ry 0 rz -90 deg; joints [-14.447, -90.117, -104.368, 14.485, 104.447, 0]
  MoveL 547 to (0, -206.4, 141.07) mm, rotated rx -90 ry 0 rz -90 deg; joints [-14.39, -90.068, -104.332, 14.4, 104.39, 0]
  MoveL 548 to (0, -205.83, 141.89) mm, rotated rx -90 ry 0 rz -90 deg; joints [-14.334, -90.019, -104.295, 14.315, 104.334, 0]
  MoveL 549 to (0, -205.26, 142.71) mm, rotated rx -90 ry 0 rz -90 deg; joints [-14.277, -89.97, -104.259, 14.23, 104.277, 0]
  MoveL 550 to (0, -204.69, 143.53) mm, rotated rx -90 ry 0 rz -90 deg; joints [-14.219, -89.922, -104.223, 14.145, 104.219, 0]
  MoveL 551 to (0, -204.12, 144.35) mm, rotated rx -90 ry 0 rz -90 deg; joints [-14.161, -89.873, -104.187, 14.06, 104.161, 0]
  MoveL 552 to (0, -203.54, 145.16) mm, rotated rx -90 ry 0 rz -90 deg; joints [-14.103, -89.824, -104.152, 13.976, 104.103, 0]
  MoveL 553 to (0, -202.96, 145.97) mm, rotated rx -90 ry 0 rz -90 deg; joints [-14.045, -89.775, -104.117, 13.892, 104.045, 0]
  MoveL 554 to (0, -202.37, 146.78) mm, rotated rx -90 ry 0 rz -90 deg; joints [-13.986, -89.726, -104.081, 13.808, 103.986, 0]
  MoveL 555 to (0, -201.78, 147.59) mm, rotated rx -90 ry 0 rz -90 deg; joints [-13.927, -89.678, -104.046, 13.724, 103.927, 0]
  MoveL 556 to (0, -201.19, 148.4) mm, rotated rx -90 ry 0 rz -90 deg; joints [-13.867, -89.629, -104.012, 13.641, 103.867, 0]
  MoveL 557 to (0, -200.6, 149.2) mm, rotated rx -90 ry 0 rz -90 deg; joints [-13.807, -89.58, -103.977, 13.558, 103.807, 0]
  MoveL 558 to (0, -200, 150) mm, rotated rx -90 ry 0 rz -90 deg; joints [-13.746, -89.532, -103.943, 13.475, 103.746, 0]
  MoveL 559 to (0, -199.4, 150.8) mm, rotated rx -90 ry 0 rz -90 deg; joints [-13.686, -89.483, -103.908, 13.392, 103.686, 0]
  MoveL 560 to (0, -198.79, 151.6) mm, rotated rx -90 ry 0 rz -90 deg; joints [-13.624, -89.435, -103.874, 13.309, 103.625, 0]
  MoveL 561 to (0, -198.19, 152.39) mm, rotated rx -90 ry 0 rz -90 deg; joints [-13.563, -89.386, -103.841, 13.227, 103.563, 0]
  MoveL 562 to (0, -197.58, 153.18) mm, rotated rx -90 ry 0 rz -90 deg; joints [-13.501, -89.338, -103.807, 13.145, 103.501, 0]
  MoveL 563 to (0, -196.96, 153.97) mm, rotated rx -90 ry 0 rz -90 deg; joints [-13.439, -89.29, -103.773, 13.063, 103.439, 0]
  MoveL 564 to (0, -196.34, 154.75) mm, rotated rx -90 ry 0 rz -90 deg; joints [-13.376, -89.241, -103.74, 12.982, 103.376, 0]
  MoveL 565 to (0, -195.72, 155.54) mm, rotated rx -90 ry 0 rz -90 deg; joints [-13.313, -89.193, -103.707, 12.9, 103.313, 0]
  MoveL 566 to (0, -195.1, 156.32) mm, rotated rx -90 ry 0 rz -90 deg; joints [-13.25, -89.145, -103.674, 12.819, 103.25, 0]
  MoveL 567 to (0, -194.48, 157.1) mm, rotated rx -90 ry 0 rz -90 deg; joints [-13.186, -89.096, -103.642, 12.738, 103.186, 0]
  MoveL 568 to (0, -193.85, 157.87) mm, rotated rx -90 ry 0 rz -90 deg; joints [-13.122, -89.048, -103.609, 12.658, 103.122, 0]
  MoveL 569 to (0, -193.21, 158.65) mm, rotated rx -90 ry 0 rz -90 deg; joints [-13.057, -89, -103.577, 12.577, 103.057, 0]
  MoveL 570 to (0, -192.58, 159.42) mm, rotated rx -90 ry 0 rz -90 deg; joints [-12.992, -88.952, -103.545, 12.497, 102.992, 0]
  MoveL 571 to (0, -191.94, 160.19) mm, rotated rx -90 ry 0 rz -90 deg; joints [-12.927, -88.904, -103.513, 12.417, 102.927, 0]
  MoveL 572 to (0, -191.3, 160.95) mm, rotated rx -90 ry 0 rz -90 deg; joints [-12.861, -88.856, -103.481, 12.337, 102.861, 0]
  MoveL 573 to (0, -190.65, 161.72) mm, rotated rx -90 ry 0 rz -90 deg; joints [-12.795, -88.808, -103.45, 12.258, 102.795, 0]
  MoveL 574 to (0, -190, 162.48) mm, rotated rx -90 ry 0 rz -90 deg; joints [-12.729, -88.76, -103.419, 12.179, 102.729, 0]
  MoveL 575 to (0, -189.35, 163.23) mm, rotated rx -90 ry 0 rz -90 deg; joints [-12.662, -88.712, -103.387, 12.1, 102.662, 0]
  MoveL 576 to (0, -188.7, 163.99) mm, rotated rx -90 ry 0 rz -90 deg; joints [-12.595, -88.665, -103.357, 12.021, 102.595, 0]
  MoveL 577 to (0, -188.04, 164.74) mm, rotated rx -90 ry 0 rz -90 deg; joints [-12.528, -88.617, -103.326, 11.943, 102.528, 0]
  MoveL 578 to (0, -187.38, 165.49) mm, rotated rx -90 ry 0 rz -90 deg; joints [-12.46, -88.569, -103.295, 11.865, 102.46, 0]
  MoveL 579 to (0, -186.72, 166.24) mm, rotated rx -90 ry 0 rz -90 deg; joints [-12.392, -88.521, -103.265, 11.787, 102.392, 0]
  MoveL 580 to (0, -186.05, 166.99) mm, rotated rx -90 ry 0 rz -90 deg; joints [-12.323, -88.474, -103.235, 11.709, 102.323, 0]
  MoveL 581 to (0, -185.38, 167.73) mm, rotated rx -90 ry 0 rz -90 deg; joints [-12.254, -88.426, -103.205, 11.632, 102.254, 0]
  MoveL 582 to (0, -184.71, 168.47) mm, rotated rx -90 ry 0 rz -90 deg; joints [-12.185, -88.379, -103.176, 11.554, 102.185, 0]
  MoveL 583 to (0, -184.04, 169.2) mm, rotated rx -90 ry 0 rz -90 deg; joints [-12.115, -88.331, -103.146, 11.478, 102.115, 0]
  MoveL 584 to (0, -183.36, 169.94) mm, rotated rx -90 ry 0 rz -90 deg; joints [-12.045, -88.284, -103.117, 11.401, 102.045, 0]
  MoveL 585 to (0, -182.68, 170.67) mm, rotated rx -90 ry 0 rz -90 deg; joints [-11.974, -88.237, -103.088, 11.324, 101.974, 0]
  MoveL 586 to (0, -182, 171.4) mm, rotated rx -90 ry 0 rz -90 deg; joints [-11.904, -88.189, -103.059, 11.248, 101.904, 0]
  MoveL 587 to (0, -181.31, 172.12) mm, rotated rx -90 ry 0 rz -90 deg; joints [-11.832, -88.142, -103.03, 11.172, 101.832, 0]
  MoveL 588 to (0, -180.62, 172.85) mm, rotated rx -90 ry 0 rz -90 deg; joints [-11.761, -88.095, -103.002, 11.097, 101.761, 0]
  MoveL 589 to (0, -179.93, 173.57) mm, rotated rx -90 ry 0 rz -90 deg; joints [-11.689, -88.048, -102.974, 11.021, 101.689, 0]
  MoveL 590 to (0, -179.23, 174.29) mm, rotated rx -90 ry 0 rz -90 deg; joints [-11.617, -88.001, -102.945, 10.946, 101.617, 0]
  MoveL 591 to (0, -178.53, 175) mm, rotated rx -90 ry 0 rz -90 deg; joints [-11.544, -87.954, -102.918, 10.872, 101.544, 0]
  MoveL 592 to (0, -177.83, 175.71) mm, rotated rx -90 ry 0 rz -90 deg; joints [-11.471, -87.907, -102.89, 10.797, 101.471, 0]
  MoveL 593 to (0, -177.13, 176.42) mm, rotated rx -90 ry 0 rz -90 deg; joints [-11.398, -87.86, -102.863, 10.723, 101.398, 0]
  MoveL 594 to (0, -176.42, 177.13) mm, rotated rx -90 ry 0 rz -90 deg; joints [-11.324, -87.813, -102.835, 10.649, 101.324, 0]
  MoveL 595 to (0, -175.71, 177.83) mm, rotated rx -90 ry 0 rz -90 deg; joints [-11.25, -87.767, -102.808, 10.575, 101.25, 0]
  MoveL 596 to (0, -175, 178.53) mm, rotated rx -90 ry 0 rz -90 deg; joints [-11.175, -87.72, -102.782, 10.501, 101.175, 0]
  MoveL 597 to (0, -174.29, 179.23) mm, rotated rx -90 ry 0 rz -90 deg; joints [-11.101, -87.673, -102.755, 10.428, 101.101, 0]
  MoveL 598 to (0, -173.57, 179.93) mm, rotated rx -90 ry 0 rz -90 deg; joints [-11.025, -87.627, -102.729, 10.355, 101.025, 0]
  MoveL 599 to (0, -172.85, 180.62) mm, rotated rx -90 ry 0 rz -90 deg; joints [-10.95, -87.58, -102.702, 10.283, 100.95, 0]
  MoveL 600 to (0, -172.12, 181.31) mm, rotated rx -90 ry 0 rz -90 deg; joints [-10.874, -87.534, -102.676, 10.21, 100.874, 0]
  MoveL 601 to (0, -171.4, 182) mm, rotated rx -90 ry 0 rz -90 deg; joints [-10.798, -87.487, -102.651, 10.138, 100.798, 0]
  MoveL 602 to (0, -170.67, 182.68) mm, rotated rx -90 ry 0 rz -90 deg; joints [-10.721, -87.441, -102.625, 10.066, 100.721, 0]
  MoveL 603 to (0, -169.94, 183.36) mm, rotated rx -90 ry 0 rz -90 deg; joints [-10.644, -87.395, -102.6, 9.994, 100.644, 0]
  MoveL 604 to (0, -169.2, 184.04) mm, rotated rx -90 ry 0 rz -90 deg; joints [-10.567, -87.349, -102.575, 9.923, 100.567, 0]
  MoveL 605 to (0, -168.47, 184.71) mm, rotated rx -90 ry 0 rz -90 deg; joints [-10.489, -87.302, -102.55, 9.852, 100.489, 0]
  MoveL 606 to (0, -167.73, 185.38) mm, rotated rx -90 ry 0 rz -90 deg; joints [-10.411, -87.256, -102.525, 9.781, 100.411, 0]
  MoveL 607 to (0, -166.99, 186.05) mm, rotated rx -90 ry 0 rz -90 deg; joints [-10.333, -87.21, -102.5, 9.711, 100.333, 0]
  MoveL 608 to (0, -166.24, 186.72) mm, rotated rx -90 ry 0 rz -90 deg; joints [-10.254, -87.165, -102.476, 9.641, 100.254, 0]
  MoveL 609 to (0, -165.49, 187.38) mm, rotated rx -90 ry 0 rz -90 deg; joints [-10.175, -87.119, -102.452, 9.571, 100.175, 0]
  MoveL 610 to (0, -164.74, 188.04) mm, rotated rx -90 ry 0 rz -90 deg; joints [-10.095, -87.073, -102.428, 9.501, 100.095, 0]
  MoveL 611 to (0, -163.99, 188.7) mm, rotated rx -90 ry 0 rz -90 deg; joints [-10.015, -87.027, -102.405, 9.432, 100.015, 0]
  MoveL 612 to (0, -163.23, 189.35) mm, rotated rx -90 ry 0 rz -90 deg; joints [-9.935, -86.982, -102.381, 9.363, 99.935, 0]
  MoveL 613 to (0, -162.48, 190) mm, rotated rx -90 ry 0 rz -90 deg; joints [-9.855, -86.936, -102.358, 9.294, 99.855, 0]
  MoveL 614 to (0, -161.72, 190.65) mm, rotated rx -90 ry 0 rz -90 deg; joints [-9.774, -86.891, -102.335, 9.225, 99.774, 0]
  MoveL 615 to (0, -160.95, 191.3) mm, rotated rx -90 ry 0 rz -90 deg; joints [-9.692, -86.845, -102.312, 9.157, 99.692, 0]
  MoveL 616 to (0, -160.19, 191.94) mm, rotated rx -90 ry 0 rz -90 deg; joints [-9.611, -86.8, -102.289, 9.089, 99.611, 0]
  MoveL 617 to (0, -159.42, 192.58) mm, rotated rx -90 ry 0 rz -90 deg; joints [-9.529, -86.755, -102.267, 9.022, 99.529, 0]
  MoveL 618 to (0, -158.65, 193.21) mm, rotated rx -90 ry 0 rz -90 deg; joints [-9.447, -86.71, -102.245, 8.954, 99.447, 0]
  MoveL 619 to (0, -157.87, 193.85) mm, rotated rx -90 ry 0 rz -90 deg; joints [-9.364, -86.664, -102.223, 8.887, 99.364, 0]
  MoveL 620 to (0, -157.1, 194.48) mm, rotated rx -90 ry 0 rz -90 deg; joints [-9.281, -86.619, -102.201, 8.821, 99.281, 0]
  MoveL 621 to (0, -156.32, 195.1) mm, rotated rx -90 ry 0 rz -90 deg; joints [-9.198, -86.574, -102.18, 8.754, 99.198, 0]
  MoveL 622 to (0, -155.54, 195.72) mm, rotated rx -90 ry 0 rz -90 deg; joints [-9.114, -86.53, -102.158, 8.688, 99.114, 0]
  MoveL 623 to (0, -154.75, 196.34) mm, rotated rx -90 ry 0 rz -90 deg; joints [-9.03, -86.485, -102.137, 8.622, 99.03, 0]
  MoveL 624 to (0, -153.97, 196.96) mm, rotated rx -90 ry 0 rz -90 deg; joints [-8.945, -86.44, -102.116, 8.557, 98.946, 0]
  MoveL 625 to (0, -153.18, 197.58) mm, rotated rx -90 ry 0 rz -90 deg; joints [-8.861, -86.396, -102.096, 8.491, 98.861, 0]
  MoveL 626 to (0, -152.39, 198.19) mm, rotated rx -90 ry 0 rz -90 deg; joints [-8.776, -86.351, -102.075, 8.426, 98.776, 0]
  MoveL 627 to (0, -151.6, 198.79) mm, rotated rx -90 ry 0 rz -90 deg; joints [-8.69, -86.307, -102.055, 8.362, 98.69, 0]
  MoveL 628 to (0, -150.8, 199.4) mm, rotated rx -90 ry 0 rz -90 deg; joints [-8.605, -86.262, -102.035, 8.297, 98.605, 0]
  MoveL 629 to (0, -150, 200) mm, rotated rx -90 ry 0 rz -90 deg; joints [-8.518, -86.218, -102.015, 8.233, 98.518, 0]
  MoveL 630 to (0, -149.2, 200.6) mm, rotated rx -90 ry 0 rz -90 deg; joints [-8.432, -86.174, -101.996, 8.169, 98.432, 0]
  MoveL 631 to (0, -148.4, 201.19) mm, rotated rx -90 ry 0 rz -90 deg; joints [-8.345, -86.13, -101.976, 8.106, 98.345, 0]
  MoveL 632 to (0, -147.59, 201.78) mm, rotated rx -90 ry 0 rz -90 deg; joints [-8.258, -86.086, -101.957, 8.043, 98.258, 0]
  MoveL 633 to (0, -146.78, 202.37) mm, rotated rx -90 ry 0 rz -90 deg; joints [-8.171, -86.042, -101.938, 7.98, 98.171, 0]
  MoveL 634 to (0, -145.97, 202.96) mm, rotated rx -90 ry 0 rz -90 deg; joints [-8.083, -85.998, -101.92, 7.918, 98.083, 0]
  MoveL 635 to (0, -145.16, 203.54) mm, rotated rx -90 ry 0 rz -90 deg; joints [-7.995, -85.954, -101.901, 7.855, 97.995, 0]
  MoveL 636 to (0, -144.35, 204.12) mm, rotated rx -90 ry 0 rz -90 deg; joints [-7.906, -85.91, -101.883, 7.793, 97.906, 0]
  MoveL 637 to (0, -143.53, 204.69) mm, rotated rx -90 ry 0 rz -90 deg; joints [-7.817, -85.867, -101.865, 7.732, 97.817, 0]
  MoveL 638 to (0, -142.71, 205.26) mm, rotated rx -90 ry 0 rz -90 deg; joints [-7.728, -85.823, -101.847, 7.67, 97.728, 0]
  MoveL 639 to (0, -141.89, 205.83) mm, rotated rx -90 ry 0 rz -90 deg; joints [-7.639, -85.78, -101.829, 7.609, 97.639, 0]
  MoveL 640 to (0, -141.07, 206.4) mm, rotated rx -90 ry 0 rz -90 deg; joints [-7.549, -85.737, -101.812, 7.549, 97.549, 0]
  MoveL 641 to (0, -140.24, 206.96) mm, rotated rx -90 ry 0 rz -90 deg; joints [-7.459, -85.694, -101.795, 7.488, 97.459, 0]
  MoveL 642 to (0, -139.41, 207.52) mm, rotated rx -90 ry 0 rz -90 deg; joints [-7.368, -85.65, -101.778, 7.428, 97.368, 0]
  MoveL 643 to (0, -138.58, 208.08) mm, rotated rx -90 ry 0 rz -90 deg; joints [-7.278, -85.607, -101.761, 7.369, 97.278, 0]
  MoveL 644 to (0, -137.75, 208.63) mm, rotated rx -90 ry 0 rz -90 deg; joints [-7.187, -85.565, -101.745, 7.309, 97.187, 0]
  MoveL 645 to (0, -136.91, 209.18) mm, rotated rx -90 ry 0 rz -90 deg; joints [-7.095, -85.522, -101.728, 7.25, 97.095, 0]
  MoveL 646 to (0, -136.08, 209.72) mm, rotated rx -90 ry 0 rz -90 deg; joints [-7.003, -85.479, -101.712, 7.191, 97.003, 0]
  MoveL 647 to (0, -135.24, 210.26) mm, rotated rx -90 ry 0 rz -90 deg; joints [-6.911, -85.436, -101.697, 7.133, 96.911, 0]
  MoveL 648 to (0, -134.4, 210.8) mm, rotated rx -90 ry 0 rz -90 deg; joints [-6.819, -85.394, -101.681, 7.075, 96.819, 0]
  MoveL 649 to (0, -133.55, 211.34) mm, rotated rx -90 ry 0 rz -90 deg; joints [-6.726, -85.351, -101.666, 7.017, 96.726, 0]
  MoveL 650 to (0, -132.71, 211.87) mm, rotated rx -90 ry 0 rz -90 deg; joints [-6.633, -85.309, -101.65, 6.96, 96.633, 0]
  MoveL 651 to (0, -131.86, 212.4) mm, rotated rx -90 ry 0 rz -90 deg; joints [-6.54, -85.267, -101.635, 6.902, 96.54, 0]
  MoveL 652 to (0, -131.01, 212.92) mm, rotated rx -90 ry 0 rz -90 deg; joints [-6.446, -85.225, -101.621, 6.846, 96.446, 0]
  MoveL 653 to (0, -130.16, 213.45) mm, rotated rx -90 ry 0 rz -90 deg; joints [-6.352, -85.183, -101.606, 6.789, 96.352, 0]
  MoveL 654 to (0, -129.3, 213.97) mm, rotated rx -90 ry 0 rz -90 deg; joints [-6.258, -85.141, -101.592, 6.733, 96.258, 0]
  MoveL 655 to (0, -128.45, 214.48) mm, rotated rx -90 ry 0 rz -90 deg; joints [-6.163, -85.099, -101.578, 6.677, 96.163, 0]
  MoveL 656 to (0, -127.59, 214.99) mm, rotated rx -90 ry 0 rz -90 deg; joints [-6.068, -85.057, -101.564, 6.621, 96.068, 0]
  MoveL 657 to (0, -126.73, 215.5) mm, rotated rx -90 ry 0 rz -90 deg; joints [-5.973, -85.016, -101.55, 6.566, 95.973, 0]
  MoveL 658 to (0, -125.86, 216.01) mm, rotated rx -90 ry 0 rz -90 deg; joints [-5.877, -84.974, -101.537, 6.511, 95.877, 0]
  MoveL 659 to (0, -125, 216.51) mm, rotated rx -90 ry 0 rz -90 deg; joints [-5.781, -84.933, -101.524, 6.457, 95.781, 0]
  MoveL 660 to (0, -124.13, 217) mm, rotated rx -90 ry 0 rz -90 deg; joints [-5.685, -84.892, -101.511, 6.403, 95.685, 0]
  MoveL 661 to (0, -123.27, 217.5) mm, rotated rx -90 ry 0 rz -90 deg; joints [-5.589, -84.85, -101.498, 6.349, 95.589, 0]
  MoveL 662 to (0, -122.39, 217.99) mm, rotated rx -90 ry 0 rz -90 deg; joints [-5.492, -84.809, -101.486, 6.295, 95.492, 0]
  MoveL 663 to (0, -121.52, 218.48) mm, rotated rx -90 ry 0 rz -90 deg; joints [-5.395, -84.769, -101.474, 6.242, 95.395, 0]
  MoveL 664 to (0, -120.65, 218.96) mm, rotated rx -90 ry 0 rz -90 deg; joints [-5.297, -84.728, -101.462, 6.189, 95.297, 0]
  MoveL 665 to (0, -119.77, 219.44) mm, rotated rx -90 ry 0 rz -90 deg; joints [-5.199, -84.687, -101.45, 6.137, 95.2, 0]
  MoveL 666 to (0, -118.89, 219.92) mm, rotated rx -90 ry 0 rz -90 deg; joints [-5.101, -84.646, -101.438, 6.085, 95.101, 0]
  MoveL 667 to (0, -118.01, 220.39) mm, rotated rx -90 ry 0 rz -90 deg; joints [-5.003, -84.606, -101.427, 6.033, 95.003, 0]
  MoveL 668 to (0, -117.13, 220.86) mm, rotated rx -90 ry 0 rz -90 deg; joints [-4.905, -84.566, -101.416, 5.981, 94.905, 0]
  MoveL 669 to (0, -116.25, 221.33) mm, rotated rx -90 ry 0 rz -90 deg; joints [-4.806, -84.525, -101.405, 5.93, 94.806, 0]
  MoveL 670 to (0, -115.36, 221.79) mm, rotated rx -90 ry 0 rz -90 deg; joints [-4.706, -84.485, -101.394, 5.879, 94.706, 0]
  MoveL 671 to (0, -114.48, 222.25) mm, rotated rx -90 ry 0 rz -90 deg; joints [-4.607, -84.445, -101.384, 5.829, 94.607, 0]
  MoveL 672 to (0, -113.59, 222.71) mm, rotated rx -90 ry 0 rz -90 deg; joints [-4.507, -84.405, -101.373, 5.779, 94.507, 0]
  MoveL 673 to (0, -112.7, 223.16) mm, rotated rx -90 ry 0 rz -90 deg; joints [-4.407, -84.365, -101.363, 5.729, 94.407, 0]
  MoveL 674 to (0, -111.8, 223.61) mm, rotated rx -90 ry 0 rz -90 deg; joints [-4.307, -84.326, -101.354, 5.68, 94.307, 0]
  MoveL 675 to (0, -110.91, 224.05) mm, rotated rx -90 ry 0 rz -90 deg; joints [-4.206, -84.286, -101.344, 5.63, 94.206, 0]
  MoveL 676 to (0, -110.01, 224.49) mm, rotated rx -90 ry 0 rz -90 deg; joints [-4.105, -84.247, -101.335, 5.582, 94.105, 0]
  MoveL 677 to (0, -109.11, 224.93) mm, rotated rx -90 ry 0 rz -90 deg; joints [-4.004, -84.208, -101.326, 5.533, 94.004, 0]
  MoveL 678 to (0, -108.21, 225.37) mm, rotated rx -90 ry 0 rz -90 deg; joints [-3.902, -84.168, -101.317, 5.485, 93.902, 0]
  MoveL 679 to (0, -107.31, 225.8) mm, rotated rx -90 ry 0 rz -90 deg; joints [-3.8, -84.129, -101.308, 5.438, 93.8, 0]
  MoveL 680 to (0, -106.41, 226.22) mm, rotated rx -90 ry 0 rz -90 deg; joints [-3.698, -84.09, -101.3, 5.39, 93.698, 0]
  MoveL 681 to (0, -105.5, 226.65) mm, rotated rx -90 ry 0 rz -90 deg; joints [-3.596, -84.052, -101.292, 5.343, 93.596, 0]
  MoveL 682 to (0, -104.6, 227.07) mm, rotated rx -90 ry 0 rz -90 deg; joints [-3.493, -84.013, -101.284, 5.297, 93.493, 0]
  MoveL 683 to (0, -103.69, 227.48) mm, rotated rx -90 ry 0 rz -90 deg; joints [-3.39, -83.974, -101.276, 5.25, 93.39, 0]
  MoveL 684 to (0, -102.78, 227.9) mm, rotated rx -90 ry 0 rz -90 deg; joints [-3.287, -83.936, -101.268, 5.205, 93.287, 0]
  MoveL 685 to (0, -101.87, 228.31) mm, rotated rx -90 ry 0 rz -90 deg; joints [-3.184, -83.898, -101.261, 5.159, 93.184, 0]
  MoveL 686 to (0, -100.95, 228.71) mm, rotated rx -90 ry 0 rz -90 deg; joints [-3.08, -83.86, -101.254, 5.114, 93.08, 0]
  MoveL 687 to (0, -100.04, 229.11) mm, rotated rx -90 ry 0 rz -90 deg; joints [-2.976, -83.822, -101.247, 5.069, 92.976, 0]
  MoveL 688 to (0, -99.12, 229.51) mm, rotated rx -90 ry 0 rz -90 deg; joints [-2.872, -83.784, -101.241, 5.024, 92.872, 0]
  MoveL 689 to (0, -98.2, 229.9) mm, rotated rx -90 ry 0 rz -90 deg; joints [-2.767, -83.746, -101.234, 4.98, 92.767, 0]
  MoveL 690 to (0, -97.28, 230.3) mm, rotated rx -90 ry 0 rz -90 deg; joints [-2.662, -83.708, -101.228, 4.937, 92.662, 0]
  MoveL 691 to (0, -96.36, 230.68) mm, rotated rx -90 ry 0 rz -90 deg; joints [-2.557, -83.671, -101.222, 4.893, 92.557, 0]
  MoveL 692 to (0, -95.44, 231.07) mm, rotated rx -90 ry 0 rz -90 deg; joints [-2.452, -83.634, -101.217, 4.85, 92.452, 0]
  MoveL 693 to (0, -94.52, 231.44) mm, rotated rx -90 ry 0 rz -90 deg; joints [-2.346, -83.596, -101.211, 4.808, 92.346, 0]
  MoveL 694 to (0, -93.59, 231.82) mm, rotated rx -90 ry 0 rz -90 deg; joints [-2.241, -83.559, -101.206, 4.765, 92.241, 0]
  MoveL 695 to (0, -92.66, 232.19) mm, rotated rx -90 ry 0 rz -90 deg; joints [-2.135, -83.522, -101.201, 4.723, 92.135, 0]
  MoveL 696 to (0, -91.73, 232.56) mm, rotated rx -90 ry 0 rz -90 deg; joints [-2.028, -83.486, -101.196, 4.682, 92.028, 0]
  MoveL 697 to (0, -90.8, 232.93) mm, rotated rx -90 ry 0 rz -90 deg; joints [-1.922, -83.449, -101.192, 4.641, 91.922, 0]
  MoveL 698 to (0, -89.87, 233.29) mm, rotated rx -90 ry 0 rz -90 deg; joints [-1.815, -83.412, -101.187, 4.6, 91.815, 0]
  MoveL 699 to (0, -88.94, 233.64) mm, rotated rx -90 ry 0 rz -90 deg; joints [-1.708, -83.376, -101.183, 4.559, 91.708, 0]
  MoveL 700 to (0, -88, 234) mm, rotated rx -90 ry 0 rz -90 deg; joints [-1.6, -83.34, -101.179, 4.519, 91.6, 0]
  MoveL 701 to (0, -87.07, 234.35) mm, rotated rx -90 ry 0 rz -90 deg; joints [-1.493, -83.304, -101.176, 4.48, 91.493, 0]
  MoveL 702 to (0, -86.13, 234.69) mm, rotated rx -90 ry 0 rz -90 deg; joints [-1.385, -83.268, -101.172, 4.44, 91.385, 0]
  MoveL 703 to (0, -85.19, 235.04) mm, rotated rx -90 ry 0 rz -90 deg; joints [-1.277, -83.232, -101.169, 4.401, 91.277, 0]
  MoveL 704 to (0, -84.25, 235.38) mm, rotated rx -90 ry 0 rz -90 deg; joints [-1.169, -83.196, -101.166, 4.363, 91.169, 0]
  MoveL 705 to (0, -83.31, 235.71) mm, rotated rx -90 ry 0 rz -90 deg; joints [-1.06, -83.161, -101.164, 4.324, 91.06, 0]
  MoveL 706 to (0, -82.37, 236.04) mm, rotated rx -90 ry 0 rz -90 deg; joints [-0.951, -83.125, -101.161, 4.287, 90.951, 0]
  MoveL 707 to (0, -81.42, 236.37) mm, rotated rx -90 ry 0 rz -90 deg; joints [-0.842, -83.09, -101.159, 4.249, 90.842, 0]
  MoveL 708 to (0, -80.48, 236.69) mm, rotated rx -90 ry 0 rz -90 deg; joints [-0.733, -83.055, -101.157, 4.212, 90.733, 0]
  MoveL 709 to (0, -79.53, 237.01) mm, rotated rx -90 ry 0 rz -90 deg; joints [-0.624, -83.02, -101.155, 4.175, 90.624, 0]
  MoveL 710 to (0, -78.58, 237.33) mm, rotated rx -90 ry 0 rz -90 deg; joints [-0.514, -82.985, -101.154, 4.139, 90.514, 0]
  MoveL 711 to (0, -77.63, 237.64) mm, rotated rx -90 ry 0 rz -90 deg; joints [-0.404, -82.951, -101.152, 4.103, 90.404, 0]
  MoveL 712 to (0, -76.68, 237.95) mm, rotated rx -90 ry 0 rz -90 deg; joints [-0.294, -82.916, -101.151, 4.067, 90.294, 0]
  MoveL 713 to (0, -75.73, 238.25) mm, rotated rx -90 ry 0 rz -90 deg; joints [-0.184, -82.882, -101.15, 4.032, 90.184, 0]
  MoveL 714 to (0, -74.78, 238.55) mm, rotated rx -90 ry 0 rz -90 deg; joints [-0.073, -82.848, -101.15, 3.998, 90.073, 0]
  MoveL 715 to (0, -73.83, 238.85) mm, rotated rx -90 ry 0 rz -90 deg; joints [0.038, -82.814, -101.149, 3.963, 89.962, 0]
  MoveL 716 to (0, -72.87, 239.14) mm, rotated rx -90 ry 0 rz -90 deg; joints [0.149, -82.78, -101.149, 3.929, 89.851, 0]
  MoveL 717 to (0, -71.91, 239.43) mm, rotated rx -90 ry 0 rz -90 deg; joints [0.26, -82.746, -101.149, 3.895, 89.74, 0]
  MoveL 718 to (0, -70.96, 239.72) mm, rotated rx -90 ry 0 rz -90 deg; joints [0.371, -82.713, -101.149, 3.862, 89.629, 0]
  MoveL 719 to (0, -70, 240) mm, rotated rx -90 ry 0 rz -90 deg; joints [0.483, -82.679, -101.15, 3.829, 89.517, 0]
  MoveL 720 to (0, -69.04, 240.28) mm, rotated rx -90 ry 0 rz -90 deg; joints [0.595, -82.646, -101.151, 3.797, 89.405, 0]
  MoveL 721 to (0, -68.08, 240.55) mm, rotated rx -90 ry 0 rz -90 deg; joints [0.707, -82.613, -101.152, 3.765, 89.293, 0]
  MoveL 722 to (0, -67.11, 240.82) mm, rotated rx -90 ry 0 rz -90 deg; joints [0.819, -82.58, -101.153, 3.733, 89.181, 0]
  MoveL 723 to (0, -66.15, 241.09) mm, rotated rx -90 ry 0 rz -90 deg; joints [0.931, -82.547, -101.154, 3.702, 89.069, 0]
  MoveL 724 to (0, -65.19, 241.35) mm, rotated rx -90 ry 0 rz -90 deg; joints [1.044, -82.515, -101.156, 3.671, 88.956, 0]
  MoveL 725 to (0, -64.22, 241.61) mm, rotated rx -90 ry 0 rz -90 deg; joints [1.157, -82.482, -101.158, 3.64, 88.843, 0]
  MoveL 726 to (0, -63.26, 241.87) mm, rotated rx -90 ry 0 rz -90 deg; joints [1.27, -82.45, -101.16, 3.61, 88.73, 0]
  MoveL 727 to (0, -62.29, 242.12) mm, rotated rx -90 ry 0 rz -90 deg; joints [1.383, -82.418, -101.162, 3.58, 88.617, 0]
  MoveL 728 to (0, -61.32, 242.36) mm, rotated rx -90 ry 0 rz -90 deg; joints [1.496, -82.386, -101.165, 3.551, 88.504, 0]
  MoveL 729 to (0, -60.35, 242.61) mm, rotated rx -90 ry 0 rz -90 deg; joints [1.61, -82.354, -101.168, 3.522, 88.39, 0]
  MoveL 730 to (0, -59.38, 242.85) mm, rotated rx -90 ry 0 rz -90 deg; joints [1.723, -82.323, -101.171, 3.493, 88.277, 0]
  MoveL 731 to (0, -58.41, 243.08) mm, rotated rx -90 ry 0 rz -90 deg; joints [1.837, -82.291, -101.174, 3.465, 88.163, 0]
  MoveL 732 to (0, -57.44, 243.31) mm, rotated rx -90 ry 0 rz -90 deg; joints [1.951, -82.26, -101.178, 3.437, 88.049, 0]
  MoveL 733 to (0, -56.46, 243.54) mm, rotated rx -90 ry 0 rz -90 deg; joints [2.066, -82.229, -101.181, 3.41, 87.934, 0]
  MoveL 734 to (0, -55.49, 243.76) mm, rotated rx -90 ry 0 rz -90 deg; joints [2.18, -82.198, -101.185, 3.383, 87.82, 0]
  MoveL 735 to (0, -54.52, 243.98) mm, rotated rx -90 ry 0 rz -90 deg; joints [2.295, -82.167, -101.189, 3.357, 87.705, 0]
  MoveL 736 to (0, -53.54, 244.2) mm, rotated rx -90 ry 0 rz -90 deg; joints [2.409, -82.137, -101.194, 3.33, 87.591, 0]
  MoveL 737 to (0, -52.56, 244.41) mm, rotated rx -90 ry 0 rz -90 deg; joints [2.524, -82.106, -101.198, 3.305, 87.476, 0]
  MoveL 738 to (0, -51.59, 244.62) mm, rotated rx -90 ry 0 rz -90 deg; joints [2.639, -82.076, -101.203, 3.279, 87.361, 0]
  MoveL 739 to (0, -50.61, 244.82) mm, rotated rx -90 ry 0 rz -90 deg; joints [2.755, -82.046, -101.208, 3.254, 87.245, 0]
  MoveL 740 to (0, -49.63, 245.02) mm, rotated rx -90 ry 0 rz -90 deg; joints [2.87, -82.016, -101.214, 3.23, 87.13, 0]
  MoveL 741 to (0, -48.65, 245.22) mm, rotated rx -90 ry 0 rz -90 deg; joints [2.986, -81.986, -101.219, 3.205, 87.014, 0]
  MoveL 742 to (0, -47.67, 245.41) mm, rotated rx -90 ry 0 rz -90 deg; joints [3.101, -81.957, -101.225, 3.182, 86.899, 0]
  MoveL 743 to (0, -46.69, 245.6) mm, rotated rx -90 ry 0 rz -90 deg; joints [3.217, -81.927, -101.231, 3.158, 86.783, 0]
  MoveL 744 to (0, -45.71, 245.79) mm, rotated rx -90 ry 0 rz -90 deg; joints [3.333, -81.898, -101.237, 3.135, 86.667, 0]
  MoveL 745 to (0, -44.72, 245.97) mm, rotated rx -90 ry 0 rz -90 deg; joints [3.449, -81.869, -101.244, 3.113, 86.551, 0]
  MoveL 746 to (0, -43.74, 246.14) mm, rotated rx -90 ry 0 rz -90 deg; joints [3.566, -81.84, -101.25, 3.091, 86.434, 0]
  MoveL 747 to (0, -42.76, 246.32) mm, rotated rx -90 ry 0 rz -90 deg; joints [3.682, -81.812, -101.257, 3.069, 86.318, 0]
  MoveL 748 to (0, -41.77, 246.49) mm, rotated rx -90 ry 0 rz -90 deg; joints [3.799, -81.783, -101.264, 3.048, 86.201, 0]
  MoveL 749 to (0, -40.79, 246.65) mm, rotated rx -90 ry 0 rz -90 deg; joints [3.915, -81.755, -101.272, 3.027, 86.085, 0]
  MoveL 750 to (0, -39.8, 246.81) mm, rotated rx -90 ry 0 rz -90 deg; joints [4.032, -81.727, -101.279, 3.006, 85.968, 0]
  MoveL 751 to (0, -38.81, 246.97) mm, rotated rx -90 ry 0 rz -90 deg; joints [4.149, -81.699, -101.287, 2.986, 85.851, 0]
  MoveL 752 to (0, -37.83, 247.12) mm, rotated rx -90 ry 0 rz -90 deg; joints [4.266, -81.671, -101.295, 2.966, 85.734, 0]
  MoveL 753 to (0, -36.84, 247.27) mm, rotated rx -90 ry 0 rz -90 deg; joints [4.383, -81.643, -101.304, 2.947, 85.617, 0]
  MoveL 754 to (0, -35.85, 247.42) mm, rotated rx -90 ry 0 rz -90 deg; joints [4.501, -81.616, -101.312, 2.928, 85.499, 0]
  MoveL 755 to (0, -34.86, 247.56) mm, rotated rx -90 ry 0 rz -90 deg; joints [4.618, -81.589, -101.321, 2.91, 85.382, 0]
  MoveL 756 to (0, -33.87, 247.7) mm, rotated rx -90 ry 0 rz -90 deg; joints [4.736, -81.562, -101.33, 2.892, 85.265, 0]
  MoveL 757 to (0, -32.88, 247.83) mm, rotated rx -90 ry 0 rz -90 deg; joints [4.853, -81.535, -101.339, 2.874, 85.147, 0]
  MoveL 758 to (0, -31.89, 247.96) mm, rotated rx -90 ry 0 rz -90 deg; joints [4.971, -81.508, -101.349, 2.857, 85.029, 0]
  MoveL 759 to (0, -30.9, 248.08) mm, rotated rx -90 ry 0 rz -90 deg; joints [5.089, -81.482, -101.358, 2.84, 84.911, 0]
  MoveL 760 to (0, -29.91, 248.2) mm, rotated rx -90 ry 0 rz -90 deg; joints [5.207, -81.456, -101.368, 2.824, 84.793, 0]
  MoveL 761 to (0, -28.91, 248.32) mm, rotated rx -90 ry 0 rz -90 deg; joints [5.325, -81.43, -101.378, 2.808, 84.675, 0]
  MoveL 762 to (0, -27.92, 248.44) mm, rotated rx -90 ry 0 rz -90 deg; joints [5.443, -81.404, -101.388, 2.792, 84.557, 0]
  MoveL 763 to (0, -26.93, 248.55) mm, rotated rx -90 ry 0 rz -90 deg; joints [5.561, -81.378, -101.399, 2.777, 84.439, 0]
  MoveL 764 to (0, -25.93, 248.65) mm, rotated rx -90 ry 0 rz -90 deg; joints [5.68, -81.353, -101.41, 2.762, 84.32, 0]
  MoveL 765 to (0, -24.94, 248.75) mm, rotated rx -90 ry 0 rz -90 deg; joints [5.798, -81.327, -101.421, 2.748, 84.202, 0]
  MoveL 766 to (0, -23.94, 248.85) mm, rotated rx -90 ry 0 rz -90 deg; joints [5.917, -81.302, -101.432, 2.734, 84.083, 0]
  MoveL 767 to (0, -22.95, 248.94) mm, rotated rx -90 ry 0 rz -90 deg; joints [6.035, -81.277, -101.444, 2.721, 83.965, 0]
  MoveL 768 to (0, -21.95, 249.03) mm, rotated rx -90 ry 0 rz -90 deg; joints [6.154, -81.253, -101.455, 2.708, 83.846, 0]
  MoveL 769 to (0, -20.96, 249.12) mm, rotated rx -90 ry 0 rz -90 deg; joints [6.273, -81.228, -101.467, 2.695, 83.727, 0]
  MoveL 770 to (0, -19.96, 249.2) mm, rotated rx -90 ry 0 rz -90 deg; joints [6.392, -81.204, -101.479, 2.683, 83.608, 0]
  MoveL 771 to (0, -18.97, 249.28) mm, rotated rx -90 ry 0 rz -90 deg; joints [6.51, -81.18, -101.492, 2.671, 83.49, 0]
  MoveL 772 to (0, -17.97, 249.35) mm, rotated rx -90 ry 0 rz -90 deg; joints [6.629, -81.156, -101.504, 2.66, 83.371, 0]
  MoveL 773 to (0, -16.97, 249.42) mm, rotated rx -90 ry 0 rz -90 deg; joints [6.749, -81.132, -101.517, 2.649, 83.251, 0]
  MoveL 774 to (0, -15.98, 249.49) mm, rotated rx -90 ry 0 rz -90 deg; joints [6.868, -81.108, -101.53, 2.638, 83.132, 0]
  MoveL 775 to (0, -14.98, 249.55) mm, rotated rx -90 ry 0 rz -90 deg; joints [6.987, -81.085, -101.543, 2.628, 83.013, 0]
  MoveL 776 to (0, -13.98, 249.61) mm, rotated rx -90 ry 0 rz -90 deg; joints [7.106, -81.062, -101.557, 2.619, 82.894, 0]
  MoveL 777 to (0, -12.98, 249.66) mm, rotated rx -90 ry 0 rz -90 deg; joints [7.225, -81.039, -101.57, 2.609, 82.775, 0]
  MoveL 778 to (0, -11.99, 249.71) mm, rotated rx -90 ry 0 rz -90 deg; joints [7.345, -81.016, -101.584, 2.601, 82.655, 0]
  MoveL 779 to (0, -10.99, 249.76) mm, rotated rx -90 ry 0 rz -90 deg; joints [7.464, -80.994, -101.599, 2.592, 82.536, 0]
